Omron Sysmac Studio project ProjFinal (Sysmac Studio 1.56.0.64011, StandardProject)
(* A implementar Expedição *)

# Controller new_Controller_0: NX1P2-1040DT1 version 1.60
Units and slaves: Unit 1 : NX-ID5442 (N1); Unit 2 : NX-OD5256 (N2)
Task PrimaryTask (priority 4, period or condition 2000): Program0
Library OEN_Communication_V1_0_22 1.0.22 (contents left out)

VAR_GLOBAL
    Garra_LIDAzul_Apertar : BOOL;  (* Outputs *)
    out_dig : ARRAY[0..99] OF BOOL;
    in_dig : ARRAY[0..99] OF BOOL;
    out_analog : ARRAY[0..99] OF WORD;  (* [2] Eixo_X_Verde *)
    inp_analog : ARRAY[0..99] OF WORD;
    Requests : ARRAY[0..3] OF OEN\Modbus\sModbusReq := [(Enable := True, NodeAdr := 1, FunctionCode := Fn02_ReadDiscreteInputs, Read := (StartAddressRemote := 0, StartAddressLocal := 0, Count := 90), Write := (StartAddressRemote := 0, StartAddressLocal := 0, Count := 100)), (Enable := True, NodeAdr := 1, FunctionCode := Fn15_WriteMultipleCoils, Read := (StartAddressRemote := 0, StartAddressLocal := 0, Count := 100), Write := (StartAddressRemote := 0, StartAddressLocal := 0, Count := 95)), (Enable := True, NodeAdr := 1, FunctionCode := Fn04_ReadInputRegisters, Read := (StartAddressRemote := 0, StartAddressLocal := 0, Count := 50), Write := (StartAddressRemote := 0, StartAddressLocal := 0, Count := 100)), (Enable := True, NodeAdr := 1, FunctionCode := Fn16_WriteMultipleRegisters, Read := (StartAddressRemote := 0, StartAddressLocal := 0, Count := 0), Write := (StartAddressRemote := 0, StartAddressLocal := 0, Count := 50))];
END_VAR
VAR_GLOBAL RETAIN
    Sensor_X_Inicial AT %D33.05 : BOOL;  (* Inputs *)
    Passadeira_2_BaseVerde AT %D18.03 : BOOL;  (* Outputs *)
    Eixo_X_LIDVerde AT %D17.07 : BOOL;  (* Outputs *)
    Sensor_Z_LID_Verde AT %D9.00 : BOOL;  (* Inputs *)
    Botao_START AT %D7.00 : BOOL;  (* Inputs *)
    Botao_RESET AT %D7.02 : BOOL;  (* Inputs *)
END_VAR
VAR_GLOBAL
    Botao_Emergencia : BOOL;  (* Inputs *)
END_VAR
VAR_GLOBAL RETAIN
    Botao_STOP AT %D7.01 : BOOL;  (* Inputs *)
    Sensor_Presença_Inicial AT %D33.00 : BOOL;  (* Inputs *)
    Sensor_Garra_Apertar_Inicial AT %D33.07 : BOOL;  (* Inputs *)
    Sensor_Garra_Levantar_Inicial AT %D33.08 : BOOL;  (* Inputs *)
    Sensor_Succao_Inicial AT %D33.03 : BOOL;  (* Inputs *)
    Sensor_Rodar_Inicial AT %D33.04 : BOOL;  (* Inputs *)
END_VAR
VAR_GLOBAL
    Sensor_LIDS_Inicial : BOOL;  (* Inputs *)
END_VAR
VAR_GLOBAL RETAIN
    Sensor_CNC AT %D33.02 : BOOL;  (* Inputs *)
    Sensor_Presenca_LIDS_Geral AT %D33.01 : BOOL;  (* Inputs *)
END_VAR
VAR_GLOBAL
    Sensor_Presenca_LIDS_Verde : BOOL;  (* Inputs *)
    Sensor_Presenca_LIDS_Azul : BOOL;  (* Inputs *)
END_VAR
VAR_GLOBAL RETAIN
    Sensor_Garra_Apertar_LID_Azul AT %D8.01 : BOOL;  (* Inputs *)
    Sensor_Garra_Apertar_LID_Verde AT %D8.00 : BOOL;  (* Inputs *)
    Fim_Curso_Garra_LID_Verde AT %D8.02 : BOOL;  (* Inputs *)
    Fim_Curso_Garra_LID_Azul AT %D8.03 : BOOL;  (* Inputs *)
    Sensor_Z_LID_Azul AT %D9.01 : BOOL;  (* Inputs *)
    Sensor_X_LID_Verde AT %D9.02 : BOOL;  (* Inputs *)
    Sensor_X_LID_Azul AT %D9.03 : BOOL;  (* Inputs *)
    Sensor_Succao_LID_Verde AT %D9.04 : BOOL;  (* Inputs *)
    Sensor_Succao_LID_Azul AT %D9.05 : BOOL;  (* Inputs *)
    Sensor_Rodar_Gripper_LID_Verde AT %D9.06 : BOOL;  (* Inputs *)
    Sensor_Rodar_Gripper_LID_Azul AT %D9.07 : BOOL;  (* Inputs *)
    Sensor_Rodar_LID_Verde AT %D9.08 : BOOL;  (* Inputs *)
    Sensor_Rodar_LID_Azul AT %D9.09 : BOOL;  (* Inputs *)
END_VAR
VAR_GLOBAL
    Sensor_Presenca_Integracao_LIDVerde : BOOL;  (* Inputs *)
    Sensor_Presenca_Integracao_LIDAzul : BOOL;  (* Inputs *)
    Sensor_Presenca_Bases : BOOL;  (* Inputs *)
    Sensor_Presenca_BaseVerde : BOOL;  (* Inputs *)
    Sensor_Presenca_BaseAzul : BOOL;  (* Inputs *)
END_VAR
VAR_GLOBAL RETAIN
    Sensor_Garra_Apertar_BaseVerde AT %D14.00 : BOOL;  (* Inputs *)
    Sensor_Garra_Apertar_BaseAzul AT %D14.01 : BOOL;  (* Inputs *)
    Emitter_Inicial AT %D16.00 : BOOL;  (* Outputs *)
    Passadeira_Inicial AT %D16.01 : BOOL;  (* Outputs *)
END_VAR
VAR_GLOBAL
    Luz_Emergencia : BOOL;  (* Outputs *)
END_VAR
VAR_GLOBAL RETAIN
    Garra_Inicial_Apertar AT %D16.02 : BOOL;  (* Outputs *)
    Garra_Inicial_Levantar AT %D16.03 : BOOL;  (* Outputs *)
    Succao_Inicial AT %D16.04 : BOOL;  (* Outputs *)
    Rotacao_Inicial_CW AT %D16.05 : BOOL;  (* Outputs *)
    Rotacao_Inicial_CCW AT %D16.06 : BOOL;  (* Outputs *)
    Botao_CNC AT %D16.11 : BOOL;  (* Outputs *)
END_VAR
VAR_GLOBAL
    Garra_LIDVerde_Apertar : BOOL;  (* Outputs *)
    Garra_LIDVerde_Levantar : BOOL;  (* Outputs *)
    Garra_LIDAzul_Levantar : BOOL;  (* Outputs *)
END_VAR
VAR_GLOBAL RETAIN
    Eixo_X_LIDAzul AT %D17.08 : BOOL;  (* Outputs *)
    Eixo_Z_LIDVerde AT %D17.09 : BOOL;  (* Outputs *)
    Eixo_Z_LIDAzul AT %D17.10 : BOOL;  (* Outputs *)
    Succao_LIDVerde AT %D17.11 : BOOL;  (* Outputs *)
    Succao_LIDAzul AT %D17.12 : BOOL;  (* Outputs *)
    Rodar_Gripper_LIDVerde AT %D17.13 : BOOL;  (* Outputs *)
    Rodar_Gripper_LIDAzul AT %D17.14 : BOOL;  (* Outputs *)
    Rodar_CCW_LIDVerde AT %D17.15 : BOOL;  (* Outputs *)
    Rodar_CCW_LIDAzul AT %D18.00 : BOOL;  (* Outputs *)
    Rodar_CW_LIDVerde AT %D18.01 : BOOL;  (* Outputs *)
    Rodar_CW_LIDAzul AT %D18.02 : BOOL;  (* Outputs *)
    Passadeira_2_BaseAzul AT %D18.04 : BOOL;  (* Outputs *)
    Braço_Verde AT %D19.02 : BOOL;  (* Outputs *)
    Braço_Azul AT %D19.04 : BOOL;  (* Outputs *)
    Passadeira_1_BaseVerde AT %D19.06 : BOOL;  (* Outputs *)
    Passadeira_1_BaseAzul AT %D19.07 : BOOL;  (* Outputs *)
    Garra_BaseVerde_Apertar AT %D28.00 : BOOL;  (* Outputs *)
    Garra_BaseAzul_Apertar AT %D28.01 : BOOL;  (* Outputs *)
END_VAR
VAR_GLOBAL
    Luz_LIDVerde : BOOL;  (* Outputs *)
    Luz_LIDAzul : BOOL;  (* Outputs *)
    Luz_BaseVerde : BOOL;  (* Outputs *)
    Luz_BaseAzul : BOOL;  (* Outputs *)
END_VAR
VAR_GLOBAL RETAIN
    Sensor_Z_Inicial AT %D33.06 : BOOL;  (* Inputs *)
    Eixo_X_Inicial AT %D16.07 : BOOL;  (* Outputs *)
    Eixo_Z_Inicial AT %D16.08 : BOOL;  (* Outputs *)
    Visão_Inicial AT %D10 : INT;
    Visão_LIDS AT %D11 : INT;
    Visão_Bases AT %D12 : INT;
    Passadeira_1_LIDS AT %D17.00 : BOOL;
    Passadeira_2_LIDS AT %D17.01 : BOOL;
    Passadeira_3_LIDS AT %D17.02 : BOOL;
    Passadeira_1_Geral AT %D19.00 : BOOL;
    Passadeira_2_Geral AT %D19.01 : BOOL;
    Passadeira_Braço_Verde AT %D19.03 : BOOL;
    Passadeira_Braço_Azul AT %D19.05 : BOOL;
END_VAR
VAR_GLOBAL
    Eixo_X_Verde : REAL;
    Eixo_Z_Verde : REAL;
END_VAR
VAR_GLOBAL RETAIN
    Succao_Verde AT %D28.04 : BOOL;
    Rotacao_CCW_Verde AT %D28.06 : BOOL;
    Rotacao_CW_Verde AT %D28.08 : BOOL;
END_VAR
VAR_GLOBAL
    Eixo_X_Azul : REAL;
    Eixo_Z_Azul : REAL;
END_VAR
VAR_GLOBAL RETAIN
    Succao_Azul AT %D28.05 : BOOL;
    Rotacao_CCW_Azul AT %D28.07 : BOOL;
    Rotacao_CW_Azul AT %D28.09 : BOOL;
    Sensor_Succao_Verde AT %D14.02 : BOOL;
    Sensor_Succao_Azul AT %D14.03 : BOOL;
END_VAR
VAR_GLOBAL
    Sensor_X_Verde : REAL;
    Sensor_Z_Verde : REAL;
    Sensor_X_Azul : REAL;
    Sensor_Z_Azul : REAL;
END_VAR
VAR_GLOBAL RETAIN
    Sensor_Rodar_Verde AT %D14.06 : BOOL;
    Sensor_Rodar_Azul AT %D14.07 : BOOL;
END_VAR
VAR_GLOBAL
    etapas_integração : INT;
    etapas_lids : INT;
    etapas_bases : INT;
    etapas_separaçãoinicial : INT;
    etapas_organização : INT;
    etapas_main : INT;
END_VAR
VAR_GLOBAL RETAIN
    Curva_Rolos_Verde AT %D29.04 : BOOL;
    Rolos_Verde_1 AT %D29.01 : BOOL;
    Rolos_Verde_2 AT %D29.02 : BOOL;
    Rolos_Verde_3 AT %D29.03 : BOOL;
    Garra_Direita_Verde AT %D29.07 : BOOL;
    Garra_Esquerda_Verde AT %D29.05 : BOOL;
    Levantar_Empilhador_Verde AT %D29.06 : BOOL;
    Sensor_Presença_PeçasVerdes AT %D15.00 : BOOL;
    FC_Meio_Verde AT %D15.01 : BOOL;
    FC_Esquerdo_Verde AT %D15.02 : BOOL;
    FC_Direito_Verde AT %D15.03 : BOOL;
    Sensor_Levantar_Empilhador_Verde AT %D15.04 : BOOL;
    Conta_Empi_Verde AT %D25 : INT;
    Sensor_Posição_Empi_Verde AT %D15.05 : BOOL;
END_VAR
VAR_GLOBAL
    Contador_Lid_Verde : INT;
    Contador_Base_Azul : INT;
    Contador_Base_Verde : INT;
END_VAR
VAR_GLOBAL RETAIN
    Removedor_Bases AT %D19.08 : BOOL;
END_VAR
VAR_GLOBAL
    Contador_LID_Azul : INT;
END_VAR
VAR_GLOBAL RETAIN
    Removedor_LIDS AT %D18.05 : BOOL;
END_VAR
VAR_GLOBAL
    Contador_Integradas_Verde : INT;
    Contador_Integradas_Azul : INT;
END_VAR
VAR_GLOBAL RETAIN
    Flag_LIDS_Azul : BOOL;
    Sensor_Base_Azul AT %D13.02 : BOOL;
    Sensor_Base_Verde AT %D13.01 : BOOL;
    Flag_Integração_Azul : BOOL;
    Rolos_Azul_1 AT %D29.09 : BOOL;
    Curva_Rolos_Azul AT %D29.10 : BOOL;
    Rolos_Azul_2 AT %D29.11 : BOOL;
    Rolos_Azul_3 AT %D29.12 : BOOL;
    Garra_Esquerda_Azul AT %D29.13 : BOOL;
    Garra_Direita_Azul AT %D29.14 : BOOL;
    Levantar_Empilhador_Azul AT %D29.15 : BOOL;
    Emitter_CPVerde AT %D29.00 : BOOL;
    Emitter_CPAzul AT %D29.08 : BOOL;
    Sensor_Presença_PeçasAzuis AT %D15.06 : BOOL;
    FC_Meio_Azul AT %D15.07 : BOOL;
    FC_Esquerdo_Azul AT %D15.08 : BOOL;
    FC_Direito_Azul AT %D15.09 : BOOL;
    Sensor_Levantar_Empilhador_Azul AT %D15.10 : BOOL;
    Sensor_Posicao_Empi_Azul AT %D15.11 : BOOL;
    Conta_Empi_Azul AT %D24 : INT;
    Flag_Integração_Verde : BOOL;
    Flag_LIDS_Verde : BOOL;
    Sensor_Bases AT %D13.00 : BOOL;
END_VAR
VAR_GLOBAL
    LED_Verde : BOOL;
    LED_Vermelho : BOOL;
    Flag_Botão_STOP_SI : BOOL;
    Flag_Botao_STOP_B : BOOL;
    Flag_Botao_STOP_L : BOOL;
    Flag_Botao_STOP_I : BOOL;
    Flag_Botao_Stop_O : BOOL;
    Flag_Emergência : BOOL;
    Reset_Factory : BOOL;
    IN_BIT_01 : BOOL;  (* BOTAO START; at BuiltInIO://cpu/#0/Input_Bit_01 *)
    IN_BIT_02 : BOOL;  (* BOTAO STOP; at BuiltInIO://cpu/#0/Input_Bit_02 *)
    OUT_BIT_01 : BOOL;  (* LED VERMELHO; at BuiltInIO://cpu/#0/Output_Bit_01 *)
    OUT_BIT_02 : BOOL;  (* LED VERDE; at BuiltInIO://cpu/#0/Output_Bit_02 *)
    IN_BIT_03 : BOOL;  (* BOTAO EMERGENCIA; at BuiltInIO://cpu/#0/Input_Bit_03 *)
END_VAR
VAR_GLOBAL RETAIN
    Sensor_LID_Verde AT %D8.04 : BOOL;
    Sensor_LID_Azul AT %D8.05 : BOOL;
END_VAR
VAR_GLOBAL
    Flag_Integração_LIDVerde : BOOL;
    Flag_Integração_LIDAzul : BOOL;
END_VAR
VAR_GLOBAL RETAIN
    Sensor_Garra_Apertar_IntLIDVerde AT %D14.04 : BOOL;
    Sensor_Garra_Apertar_IntLIDAzul AT %D14.05 : BOOL;
    Garra_LIDVerdeInt_apertar AT %D28.02 : BOOL;
    Garra_LIDAzulInt_apertar AT %D28.03 : BOOL;
    Garra_LIDAzul_Levant AT %D17.06 : BOOL;
    Garra_LIDVerde_Levant AT %D17.05 : BOOL;
    Garra_LIDAzul_Apert AT %D17.04 : BOOL;
    Garra_LIDVerde_Apert AT %D17.03 : BOOL;
    Expedição_Caixas_Verdes AT %D26 : INT;
    Expedição_Caixas_Azuis AT %D27 : INT;
END_VAR
VAR_GLOBAL
    etapas_expediçãoazul : INT;
    Rolos_Exp_Azul_1 : BOOL;
    Rolos_Exp_Azul_2 : BOOL;
    Remover_Exp_Azul : BOOL;
    Emitter_Exp_Azul : BOOL;
    Rolos_Exp_Azul_3 : BOOL;
    Remover_Caixa_Azul : BOOL;
    etapas_expediçãoverde : INT;
    Rolos_Exp_Verde_1 : BOOL;
    Remover_Exp_Verde : BOOL;
    Emitter_Exp_Verde : BOOL;
    Remover_Caixa_Verde : BOOL;
    Rolos_Exp_Verde_2 : BOOL;
    Levantar_Empilhador_Azul_Expedição : BOOL;
    Garra_Direita_Azul_Expedição : BOOL;
    Levantar_Empilhador_Verde_Expedição : BOOL;
    Garra_Direita_Verde_Expedição : BOOL;
END_VAR
VAR_GLOBAL RETAIN
    Stock_Azul : INT;
    Stock_Verde : INT;
    Nº_Caixas_Expedidas_Azuis AT %D22 : INT;
    Nº_Caixas_Expedidas_Verdes AT %D23 : INT;
END_VAR
VAR_GLOBAL
    Flag_Botao_Stop_EA : BOOL;
    Flag_Botao_Stop_EV : BOOL;
END_VAR
VAR_GLOBAL RETAIN
    SI_LED AT %D7.02 : BOOL;
    L_LED AT %D7.03 : BOOL;
    B_LED AT %D7.04 : BOOL;
    I_LED AT %D7.05 : BOOL;
    A_LED AT %D7.06 : BOOL;
    E_LED AT %D7.07 : BOOL;
    Peças_Integradas_Verdes_HMI AT %D20 : INT;
    Peças_Integradas_Azuis_HMI AT %D21 : INT;
    Pusher AT %D16.09 : BOOL;
    Remove_Peças_Más AT %D16.10 : BOOL;
END_VAR
VAR_GLOBAL
    FC_Traseiro_Pusher : BOOL;
END_VAR
VAR_GLOBAL RETAIN
    Eixo_X_Verde_HMI AT %D40 : INT;
    Eixo_X_Azul_HMI AT %D41 : INT;
    Eixo_Z_Verde_HMI AT %D42 : INT;
    Eixo_Z_Azul_HMI AT %D43 : INT;
END_VAR

PROGRAM Program0
VAR
    TCP_CLIENT : OEN\Modbus\ModbusTCP_Client;
    TimerIntegraçãoAzul : TON;
    TimerIntegraçãoAzul2 : TON;
    TimerIntegraçãoAzul3 : TON;
    TimerIntegraçãoAzul4 : TON;
    TimerIntegraçãoVerde : TON;
    TimerIntegraçãoVerde2 : TON;
    TimerIntegraçãoVerde3 : TON;
    TimerIntegraçãoVerde4 : TON;
    TimerSensorEmpiVerde : TON;
    TON_EMPVERDE1 : TON;
    TON_EMPVERDE2 : TON;
    TON_EMPVERDE3 : TON;
    TON_EMPVERDE4 : TON;
    TimerSensorEmpiAzul : TON;
    TON_EMPAZUL1 : TON;
    TON_EMPAZUL2 : TON;
    TON_EMPAZUL3 : TON;
    TON_EMPAZUL4 : TON;
    Timer_Gripper_Verde : TON;
    LIDVerde1 : TON;
    LIDVerde2 : TON;
    Timer_Gripper_Azul : TON;
    LIDAzul1 : TON;
    LIDAzul2 : TON;
    TimerRemovedorBases : TON;
    Timer_Base_Verde : TON;
    Timer_Base_Azul : TON;
    TimerPickNPlace : TON;
    Timer_LidVerde_Garra : TON;
    Timer_LidAzul_Garra : TON;
    TimerRemovedorLIDS : TON;
    CTUEmpiVerde : CTU;
    CTUEmpiAzul : CTU;
    CTUIntegradasVerde : CTU;
    CTUIntegradasAzul : CTU;
    CTULidVerde : CTU;
    CTULidAzul : CTU;
    CTUBaseVerde : CTU;
    CTUBaseAzul : CTU;
    Teste : TON;
    Timer_LID_Verde : TON;
    Timer_LID_Azul : TON;
    Timer_Expedição_Azul : TON;
    TON_EMPAZUL5 : TON;
    TON_EMPAZUL6 : TON;
    TON_EMPAZUL7 : TON;
    TON_EMPAZUL8 : TON;
    TON_EMPAZUL9 : TON;
    TON_EMPAZUL10 : TON;
    TON_EMPAZUL11 : TON;
    CTD_Empi_Azul : CTD;
    CTD_Restante_Exp_Azul : CTD;
    TON_EMPVERDE5 : TON;
    TON_EMPVERDE6 : TON;
    TON_EMPVERDE7 : TON;
    TON_EMPVERDE8 : TON;
    TON_EMPVERDE9 : TON;
    TON_EMPVERDE10 : TON;
    TON_EMPVERDE11 : TON;
    TON_EMPAZUL12 : TON;
    TON_EMPVERDE12 : TON;
    CTD_Stock_Azul : CTD;
    TON_COUNTERSAZUL : TON;
    TIMERFLAGS : TON;
    TRIGSUBS : R_TRIG;
    TRIGSUBS1 : R_TRIG;
    TRIGSUB2 : R_TRIG;
    TRIGLIDA1 : R_TRIG;
    TRIGLIDV1 : R_TRIG;
    TRIGBASEA1 : R_TRIG;
    TRIGBASEV1 : R_TRIG;
    TRIGINTEGRADAV1 : R_TRIG;
    TRIGINTEGRADAA1 : R_TRIG;
    TRIGEMPV1 : R_TRIG;
    TRIGEMPA1 : R_TRIG;
    TRIGSUBS2 : R_TRIG;
    TRIGEXPVERDE1 : R_TRIG;
    TRIGEXPVERDE2 : R_TRIG;
    TRIGEXPVERDE3 : R_TRIG;
END_VAR
VAR RETAIN
    Emitter_Inicial_HMI AT %D0.00 : BOOL;
    Passadeira_Inicial_HMI AT %D0.01 : BOOL;
    Garra_Inicial_Apertar_HMI AT %D0.02 : BOOL;
    Garra_Inicial_Levantar_HMI AT %D0.03 : BOOL;
    Succao_Inicial_HMI AT %D0.04 : BOOL;
    Rotação_Inicial_CW_HMI AT %D0.05 : BOOL;
    Rotacao_Inicial_CCW_HMI AT %D0.06 : BOOL;
    Eixo_X_Inicial_HMI AT %D0.07 : BOOL;
    Eixo_Z_Inicial_HMI AT %D0.08 : BOOL;
    Botao_CNC_HMI AT %D0.09 : BOOL;
    Passadeira_1_LIDS_HMI AT %D1.00 : BOOL;
    Passadeira_2_LIDS_HMI AT %D1.01 : BOOL;
    Passadeira_3_LIDS_HMI AT %D1.02 : BOOL;
    Passadeira_2_BaseVerde_HMI AT %D1.03 : BOOL;
    Passadeira_2_BaseAzul_HMI AT %D1.04 : BOOL;
    Garra_LIDVerde_Apert_HMI AT %D1.05 : BOOL;
    Garra_LIDAzul_Apert_HMI AT %D1.06 : BOOL;
    Garra_LIDVerde_Levant_HMI AT %D1.07 : BOOL;
    Garra_LIDAzul_Levant_HMI AT %D1.08 : BOOL;
    Removedor_LIDS_HMI AT %D1.09 : BOOL;
    Eixo_X_LIDVerde_HMI AT %D2.00 : BOOL;
    Eixo_X_LIDAzul_HMI AT %D2.01 : BOOL;
    Eixo_Z_LID_Verde_HMI AT %D2.02 : BOOL;
    Eixo_Z_LIDAzul_HMI AT %D2.03 : BOOL;
    Succao_LIDVerde_HMI AT %D2.04 : BOOL;
    Succao_LIDAzul_HMI AT %D2.05 : BOOL;
    Rodar_Gripper_LIDVerde_HMI AT %D2.06 : BOOL;
    Rodar_Gripper_LIDAzul_HMI AT %D2.07 : BOOL;
    Rodar_CCW_LIDVerde_HMI AT %D2.08 : BOOL;
    Rodar_CCW_LIDAzul_HMI AT %D2.09 : BOOL;
    Rodar_CW_LIDVerde_HMI AT %D2.10 : BOOL;
    Rodar_CW_LIDAzul_HMI AT %D2.11 : BOOL;
    Passadeira_1_Geral_HMI AT %D3.00 : BOOL;
    Passadeira_2_Geral_HMI AT %D3.01 : BOOL;
    Braço_Verde_HMI AT %D3.02 : BOOL;
    Passadeira_Braço_Verde_HMI AT %D3.03 : BOOL;
    Braço_Azul_HMI AT %D3.04 : BOOL;
    Passadeira_Braço_Azul_HMI AT %D3.05 : BOOL;
    Passadeira_1_BaseVerde_HMI AT %D3.06 : BOOL;
    Passadeira_1_BaseAzul_HMI AT %D3.07 : BOOL;
    Removedor_Bases_HMI AT %D3.08 : BOOL;
    Garra_BaseAzul_Apertar_HMI AT %D4.00 : BOOL;
    Garra_BaseVerde_Apertar_HMI AT %D4.01 : BOOL;
    Garra_LIDVerdeInt_apertar_HMI AT %D4.02 : BOOL;
    Garra_LIDAzulInt_apertar_HMI AT %D4.03 : BOOL;
    Succao_Verde_HMI AT %D4.04 : BOOL;
    Succao_Azul_HMI AT %D4.05 : BOOL;
    Rotacao_CCW_Verde_HMI AT %D4.06 : BOOL;
    Rotacao_CCW_Azul_HMI AT %D4.07 : BOOL;
    Rotacao_CW_Verde_HMI AT %D4.08 : BOOL;
    Rotacao_CW_Azul_HMI AT %D4.09 : BOOL;
    Emitter_CPVerde_HMI AT %D5.00 : BOOL;
    Rolos_Verde_1_HMI AT %D5.01 : BOOL;
    Rolos_Verde_2_HMI AT %D5.02 : BOOL;
    Rolos_Verde_3_HMI AT %D5.03 : BOOL;
    Curva_Rolos_Verde_HMI AT %D5.04 : BOOL;
    Emitter_CPAzul_HMI AT %D5.05 : BOOL;
    Rolos_Azul_1_HMI AT %D5.06 : BOOL;
    Curva_Rolos_Azul_HMI AT %D5.07 : BOOL;
    Rolos_Azul_2_HMI AT %D5.08 : BOOL;
    Rolos_Azul_3_HMI AT %D5.09 : BOOL;
    Garra_Esquerda_Azul_HMI AT %D6.00 : BOOL;
    Garra_Direita_Azul_HMI AT %D6.01 : BOOL;
    Levantar_Empilhador_Azul_HMI AT %D6.02 : BOOL;
    Garra_Esquerda_Verde_HMI AT %D6.03 : BOOL;
    Levantar_Empilhador_Verde_HMI AT %D6.04 : BOOL;
    Garra_Direita_Verde_HMI AT %D6.05 : BOOL;
END_VAR
VAR
    TRIGINTEGRADAA2 : R_TRIG;
    TRIGINTEGRADAV2 : R_TRIG;
    TON_Peça_Máe : TON;
    TON_Peça_Má : TON;
END_VAR
VAR RETAIN
    Pusher_HMI AT %D0.10 : BOOL;
    Remove_Peças_Más_HMI AT %D0.11 : BOOL;
END_VAR
VAR
    RESETTON : TON;
END_VAR
VAR_EXTERNAL
    Emitter_Inicial : BOOL;
    Garra_Inicial_Apertar : BOOL;
    Garra_Inicial_Levantar : BOOL;
    Braço_Azul : BOOL;
    Braço_Verde : BOOL;
    in_dig : ARRAY[0..99] OF BOOL;
    out_dig : ARRAY[0..99] OF BOOL;
    out_analog : ARRAY[0..99] OF WORD;
    Requests : ARRAY[0..3] OF OEN\Modbus\sModbusReq;
    Botao_RESET : BOOL;
    Botao_Emergencia : BOOL;
    Botao_START : BOOL;
    Botao_STOP : BOOL;
    Luz_Emergencia : BOOL;
    Passadeira_Inicial : BOOL;
    Sensor_Presença_Inicial : BOOL;
    Sensor_Garra_Apertar_Inicial : BOOL;
    Sensor_Garra_Levantar_Inicial : BOOL;
    Sensor_CNC : BOOL;
    Sensor_Succao_Inicial : BOOL;
    Sensor_Z_Inicial : BOOL;
    Sensor_X_Inicial : BOOL;
    Sensor_Rodar_Inicial : BOOL;
    Sensor_LIDS_Inicial : BOOL;
    Sensor_Presenca_LIDS_Geral : BOOL;
    Sensor_Presenca_LIDS_Verde : BOOL;
    Sensor_Presenca_LIDS_Azul : BOOL;
    Botao_CNC : BOOL;
    Sensor_Garra_Apertar_LID_Azul : BOOL;
    Sensor_Garra_Apertar_LID_Verde : BOOL;
    Fim_Curso_Garra_LID_Verde : BOOL;
    Fim_Curso_Garra_LID_Azul : BOOL;
    Sensor_Z_LID_Verde : BOOL;
    Sensor_Z_LID_Azul : BOOL;
    Sensor_X_LID_Verde : BOOL;
    Sensor_X_LID_Azul : BOOL;
    Sensor_Succao_LID_Verde : BOOL;
    Sensor_Succao_LID_Azul : BOOL;
    Sensor_Rodar_Gripper_LID_Verde : BOOL;
    Sensor_Rodar_Gripper_LID_Azul : BOOL;
    Sensor_Rodar_LID_Verde : BOOL;
    Sensor_Rodar_LID_Azul : BOOL;
    Sensor_Presenca_Integracao_LIDVerde : BOOL;
    Sensor_Presenca_Integracao_LIDAzul : BOOL;
    Sensor_Presenca_Bases : BOOL;
    Sensor_Presenca_BaseVerde : BOOL;
    Sensor_Presenca_BaseAzul : BOOL;
    Sensor_Garra_Apertar_BaseVerde : BOOL;
    Sensor_Garra_Apertar_BaseAzul : BOOL;
    Succao_Inicial : BOOL;
    Rotacao_Inicial_CW : BOOL;
    Rotacao_Inicial_CCW : BOOL;
    Eixo_Z_Inicial : BOOL;
    Eixo_X_Inicial : BOOL;
    Garra_LIDVerde_Apertar : BOOL;
    Garra_LIDAzul_Apertar : BOOL;
    Garra_LIDVerde_Levantar : BOOL;
    Garra_LIDAzul_Levantar : BOOL;
    Eixo_X_LIDVerde : BOOL;
    Eixo_X_LIDAzul : BOOL;
    Eixo_Z_LIDVerde : BOOL;
    Eixo_Z_LIDAzul : BOOL;
    Succao_LIDVerde : BOOL;
    Succao_LIDAzul : BOOL;
    Rodar_Gripper_LIDVerde : BOOL;
    Rodar_Gripper_LIDAzul : BOOL;
    Rodar_CCW_LIDVerde : BOOL;
    Rodar_CCW_LIDAzul : BOOL;
    Rodar_CW_LIDVerde : BOOL;
    Rodar_CW_LIDAzul : BOOL;
    Passadeira_2_BaseVerde : BOOL;
    Passadeira_2_BaseAzul : BOOL;
    Passadeira_1_BaseVerde : BOOL;
    Passadeira_1_BaseAzul : BOOL;
    Garra_BaseVerde_Apertar : BOOL;
    Garra_BaseAzul_Apertar : BOOL;
    Luz_LIDVerde : BOOL;
    Luz_LIDAzul : BOOL;
    Luz_BaseVerde : BOOL;
    Luz_BaseAzul : BOOL;
    Visão_Inicial : INT;
    Visão_LIDS : INT;
    Visão_Bases : INT;
    Passadeira_1_LIDS : BOOL;
    Passadeira_2_LIDS : BOOL;
    Passadeira_3_LIDS : BOOL;
    Passadeira_1_Geral : BOOL;
    Passadeira_2_Geral : BOOL;
    Passadeira_Braço_Verde : BOOL;
    Passadeira_Braço_Azul : BOOL;
    Eixo_X_Verde : REAL;
    Eixo_Z_Verde : REAL;
    Succao_Verde : BOOL;
    Rotacao_CCW_Verde : BOOL;
    Rotacao_CW_Verde : BOOL;
    Eixo_X_Azul : REAL;
    Eixo_Z_Azul : REAL;
    Succao_Azul : BOOL;
    Rotacao_CCW_Azul : BOOL;
    Rotacao_CW_Azul : BOOL;
    Sensor_Succao_Verde : BOOL;
    Sensor_Succao_Azul : BOOL;
    Sensor_X_Verde : REAL;
    Sensor_Z_Verde : REAL;
    Sensor_X_Azul : REAL;
    Sensor_Z_Azul : REAL;
    Sensor_Rodar_Verde : BOOL;
    Sensor_Rodar_Azul : BOOL;
    inp_analog : ARRAY[0..99] OF WORD;
    etapas_integração : INT;
    etapas_lids : INT;
    etapas_bases : INT;
    etapas_separaçãoinicial : INT;
    etapas_organização : INT;
    etapas_main : INT;
    Curva_Rolos_Verde : BOOL;
    Rolos_Verde_1 : BOOL;
    Rolos_Verde_2 : BOOL;
    Rolos_Verde_3 : BOOL;
    Sensor_Presença_PeçasVerdes : BOOL;
    Garra_Esquerda_Verde : BOOL;
    FC_Meio_Verde : BOOL;
    FC_Esquerdo_Verde : BOOL;
    FC_Direito_Verde : BOOL;
    Levantar_Empilhador_Verde : BOOL;
    Sensor_Levantar_Empilhador_Verde : BOOL;
    Conta_Empi_Verde : INT;
    Sensor_Posição_Empi_Verde : BOOL;
    Garra_Direita_Verde : BOOL;
    Contador_Lid_Verde : INT;
    Contador_Base_Azul : INT;
    Contador_Base_Verde : INT;
    Removedor_Bases : BOOL;
    Contador_LID_Azul : INT;
    Removedor_LIDS : BOOL;
    Contador_Integradas_Verde : INT;
    Contador_Integradas_Azul : INT;
    Flag_LIDS_Azul : BOOL;
    Sensor_Base_Azul : BOOL;
    Sensor_Base_Verde : BOOL;
    Flag_Integração_Azul : BOOL;
    Rolos_Azul_1 : BOOL;
    Curva_Rolos_Azul : BOOL;
    Rolos_Azul_2 : BOOL;
    Rolos_Azul_3 : BOOL;
    Garra_Esquerda_Azul : BOOL;
    Garra_Direita_Azul : BOOL;
    Levantar_Empilhador_Azul : BOOL;
    Emitter_CPVerde : BOOL;
    Emitter_CPAzul : BOOL;
    Sensor_Presença_PeçasAzuis : BOOL;
    FC_Meio_Azul : BOOL;
    FC_Esquerdo_Azul : BOOL;
    FC_Direito_Azul : BOOL;
    Sensor_Levantar_Empilhador_Azul : BOOL;
    Sensor_Posicao_Empi_Azul : BOOL;
    Conta_Empi_Azul : INT;
    Flag_Integração_Verde : BOOL;
    Flag_LIDS_Verde : BOOL;
    Sensor_Bases : BOOL;
    LED_Verde : BOOL;
    LED_Vermelho : BOOL;
    Flag_Botão_STOP_SI : BOOL;
    Flag_Botao_STOP_B : BOOL;
    Flag_Botao_STOP_L : BOOL;
    Flag_Botao_STOP_I : BOOL;
    Flag_Botao_Stop_O : BOOL;
    Flag_Emergência : BOOL;
    Reset_Factory : BOOL;
    OUT_BIT_02 : BOOL;
    OUT_BIT_01 : BOOL;
    IN_BIT_01 : BOOL;
    IN_BIT_02 : BOOL;
    IN_BIT_03 : BOOL;
    Sensor_LID_Verde : BOOL;
    Sensor_LID_Azul : BOOL;
    Flag_Integração_LIDVerde : BOOL;
    Flag_Integração_LIDAzul : BOOL;
    Sensor_Garra_Apertar_IntLIDVerde : BOOL;
    Sensor_Garra_Apertar_IntLIDAzul : BOOL;
    Garra_LIDVerdeInt_apertar : BOOL;
    Garra_LIDAzulInt_apertar : BOOL;
    Garra_LIDAzul_Levant : BOOL;
    Garra_LIDVerde_Levant : BOOL;
    Garra_LIDAzul_Apert : BOOL;
    Garra_LIDVerde_Apert : BOOL;
    Expedição_Caixas_Verdes : INT;
    Expedição_Caixas_Azuis : INT;
    etapas_expediçãoazul : INT;
    Rolos_Exp_Azul_1 : BOOL;
    Rolos_Exp_Azul_2 : BOOL;
    Remover_Exp_Azul : BOOL;
    Emitter_Exp_Azul : BOOL;
    Rolos_Exp_Azul_3 : BOOL;
    Remover_Caixa_Azul : BOOL;
    etapas_expediçãoverde : INT;
    Rolos_Exp_Verde_1 : BOOL;
    Remover_Exp_Verde : BOOL;
    Emitter_Exp_Verde : BOOL;
    Remover_Caixa_Verde : BOOL;
    Rolos_Exp_Verde_2 : BOOL;
    Levantar_Empilhador_Azul_Expedição : BOOL;
    Garra_Direita_Azul_Expedição : BOOL;
    Levantar_Empilhador_Verde_Expedição : BOOL;
    Garra_Direita_Verde_Expedição : BOOL;
    Stock_Azul : INT;
    Stock_Verde : INT;
    Nº_Caixas_Expedidas_Azuis : INT;
    Nº_Caixas_Expedidas_Verdes : INT;
    Flag_Botao_Stop_EA : BOOL;
    Flag_Botao_Stop_EV : BOOL;
    SI_LED : BOOL;
    L_LED : BOOL;
    B_LED : BOOL;
    I_LED : BOOL;
    A_LED : BOOL;
    E_LED : BOOL;
    Peças_Integradas_Verdes_HMI : INT;
    Peças_Integradas_Azuis_HMI : INT;
    Pusher : BOOL;
    Remove_Peças_Más : BOOL;
    FC_Traseiro_Pusher : BOOL;
    Eixo_X_Verde_HMI : INT;
    Eixo_X_Azul_HMI : INT;
    Eixo_Z_Verde_HMI : INT;
    Eixo_Z_Azul_HMI : INT;
END_VAR
VAR
    _p1 : BOOL;
    _p2 : BOOL;
    _p3 : BOOL;
    _p4 : BOOL;
    _p5 : BOOL;
    _p6 : BOOL;
    _p7 : BOOL;
    _p8 : BOOL;
    _p9 : BOOL;
    _p10 : BOOL;
    _p11 : BOOL;
    _p12 : BOOL;
    _p13 : BOOL;
    _p14 : BOOL;
    _p15 : BOOL;
END_VAR

(* Section ModBusComm: ladder, written here as Structured Text *)

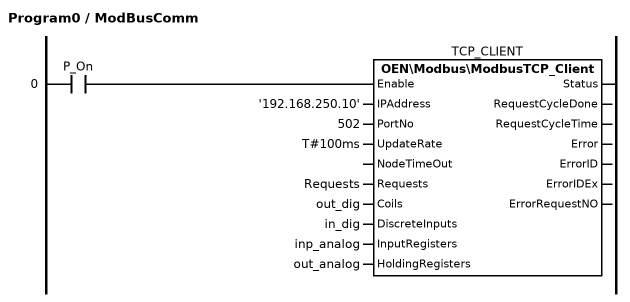
(* Rung 0 *)
TCP_CLIENT(Enable := P_On, IPAddress := '192.168.250.10', PortNo := 502, UpdateRate := T#100ms, Requests := Requests, Coils := out_dig, DiscreteInputs := in_dig, InputRegisters := inp_analog, HoldingRegisters := out_analog);

(* Section Main_Etapas: ladder, written here as Structured Text *)

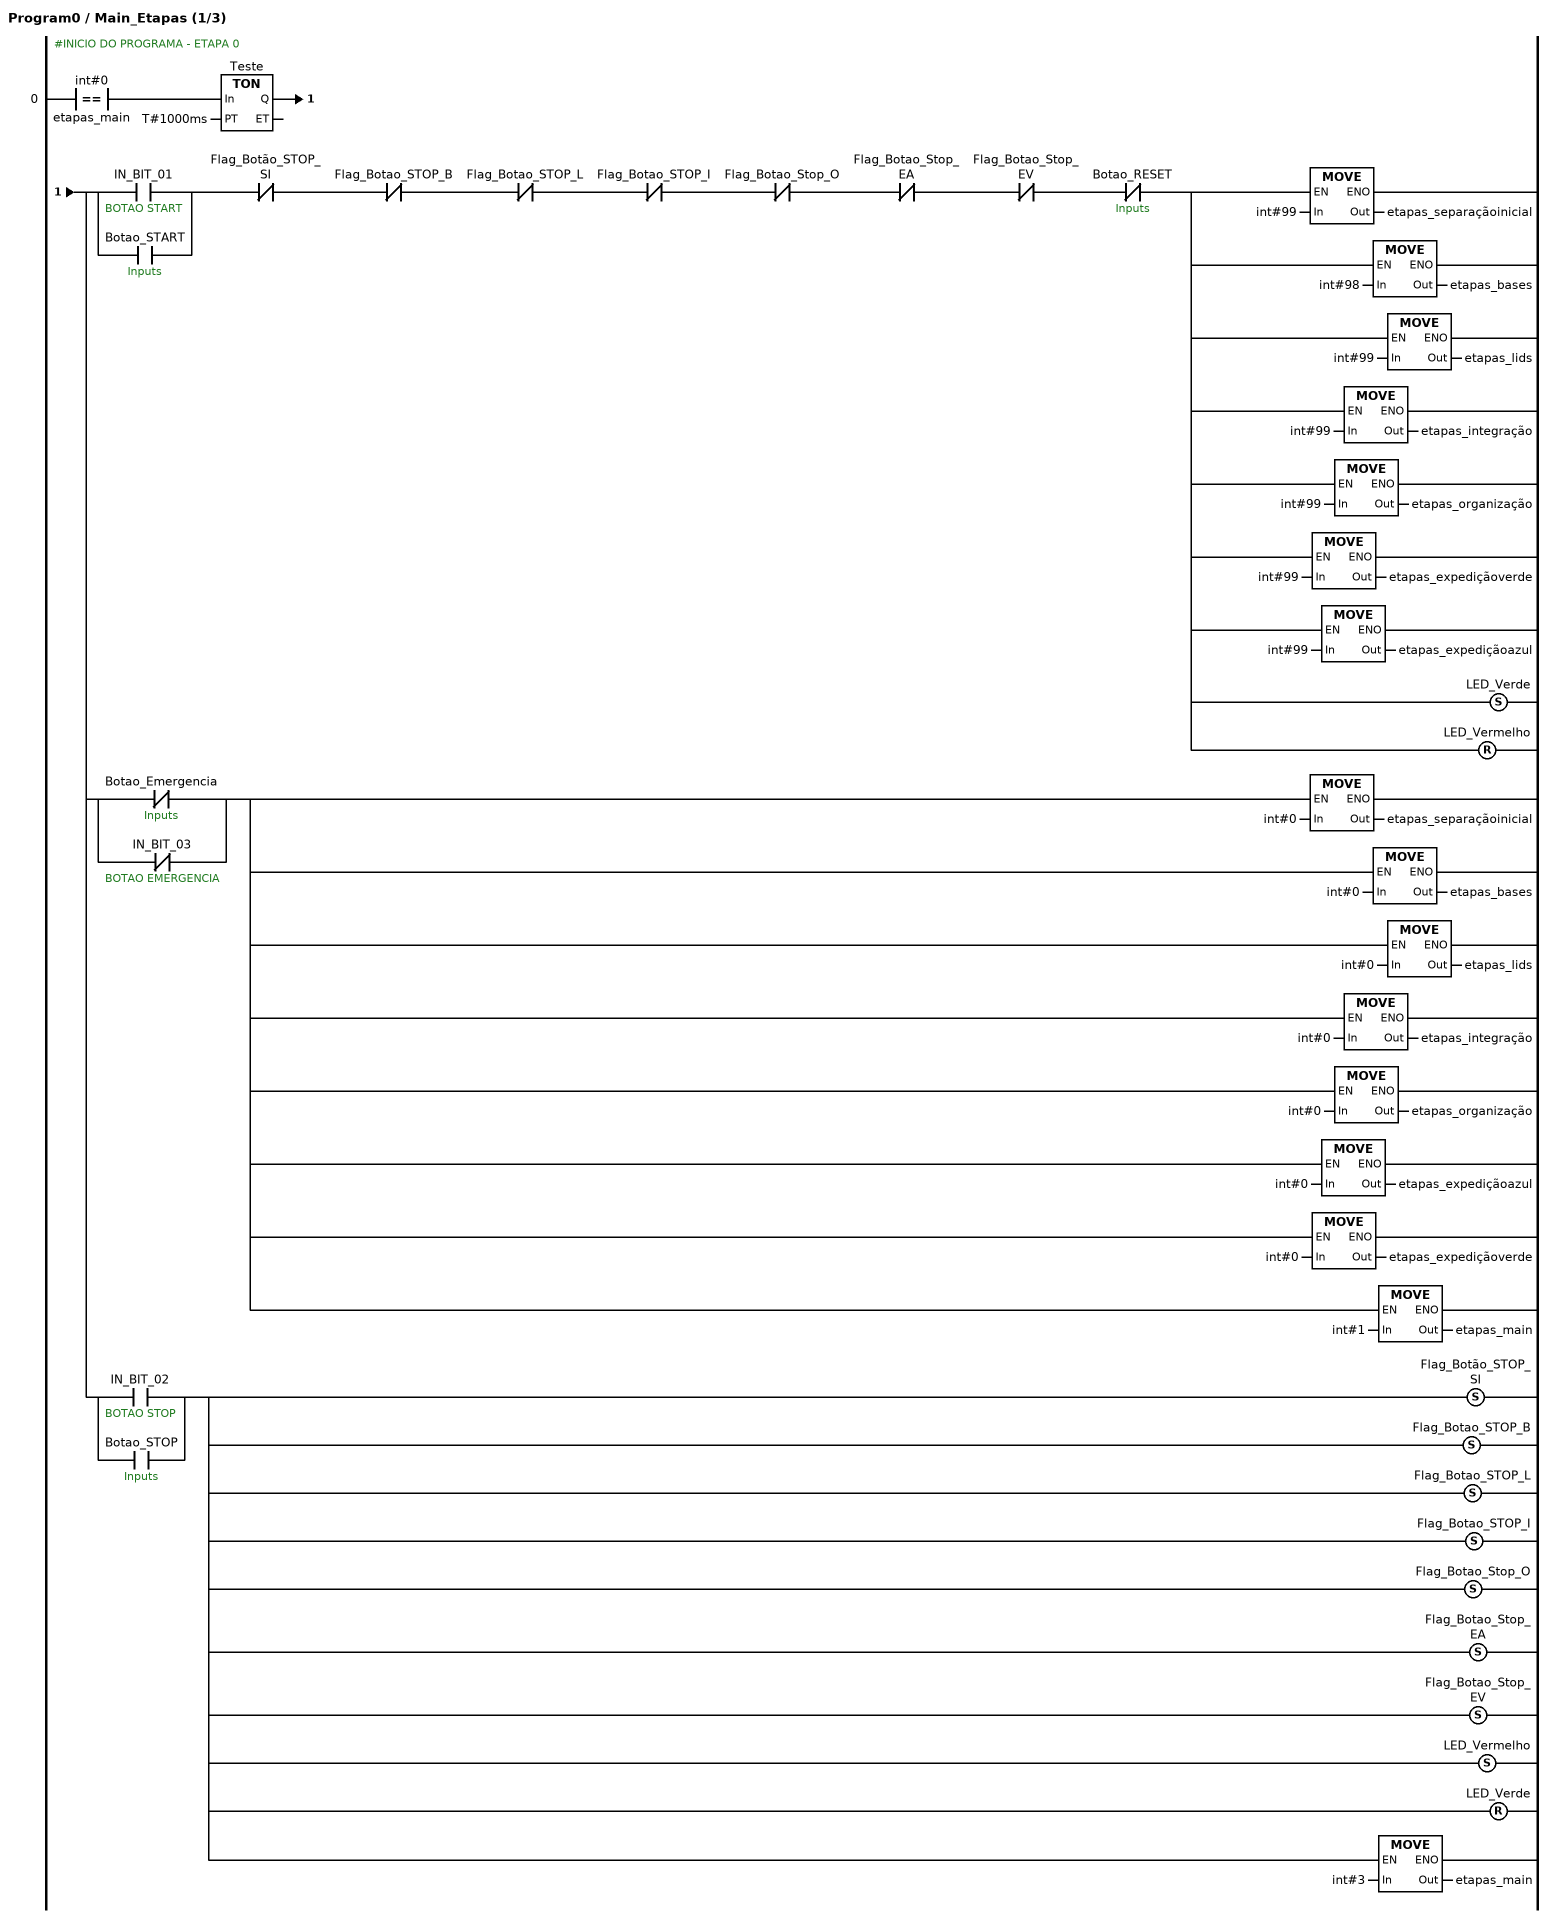
(* Rung 0: #INICIO DO PROGRAMA - ETAPA 0 *)
Teste(In := int#0 = etapas_main, PT := T#1000ms);
_p1 := Teste.Q AND (IN_BIT_01 OR Botao_START) AND NOT Flag_Botão_STOP_SI AND NOT Flag_Botao_STOP_B AND NOT Flag_Botao_STOP_L AND NOT Flag_Botao_STOP_I AND NOT Flag_Botao_Stop_O AND NOT Flag_Botao_Stop_EA AND NOT Flag_Botao_Stop_EV AND NOT Botao_RESET;
IF _p1 THEN
    etapas_separaçãoinicial := int#99;
    etapas_bases := int#98;
    etapas_lids := int#99;
    etapas_integração := int#99;
    etapas_organização := int#99;
    etapas_expediçãoverde := int#99;
    etapas_expediçãoazul := int#99;
    LED_Verde := TRUE;
    LED_Vermelho := FALSE;
END_IF;
_p2 := Teste.Q AND (NOT Botao_Emergencia OR NOT IN_BIT_03);
IF _p2 THEN
    etapas_separaçãoinicial := int#0;
    etapas_bases := int#0;
    etapas_lids := int#0;
    etapas_integração := int#0;
    etapas_organização := int#0;
    etapas_expediçãoazul := int#0;
    etapas_expediçãoverde := int#0;
    etapas_main := int#1;
END_IF;
IF Teste.Q AND (IN_BIT_02 OR Botao_STOP) THEN
    Flag_Botão_STOP_SI := TRUE;
    Flag_Botao_STOP_B := TRUE;
    Flag_Botao_STOP_L := TRUE;
    Flag_Botao_STOP_I := TRUE;
    Flag_Botao_Stop_O := TRUE;
    Flag_Botao_Stop_EA := TRUE;
    Flag_Botao_Stop_EV := TRUE;
    LED_Vermelho := TRUE;
    LED_Verde := FALSE;
    etapas_main := int#3;
END_IF;

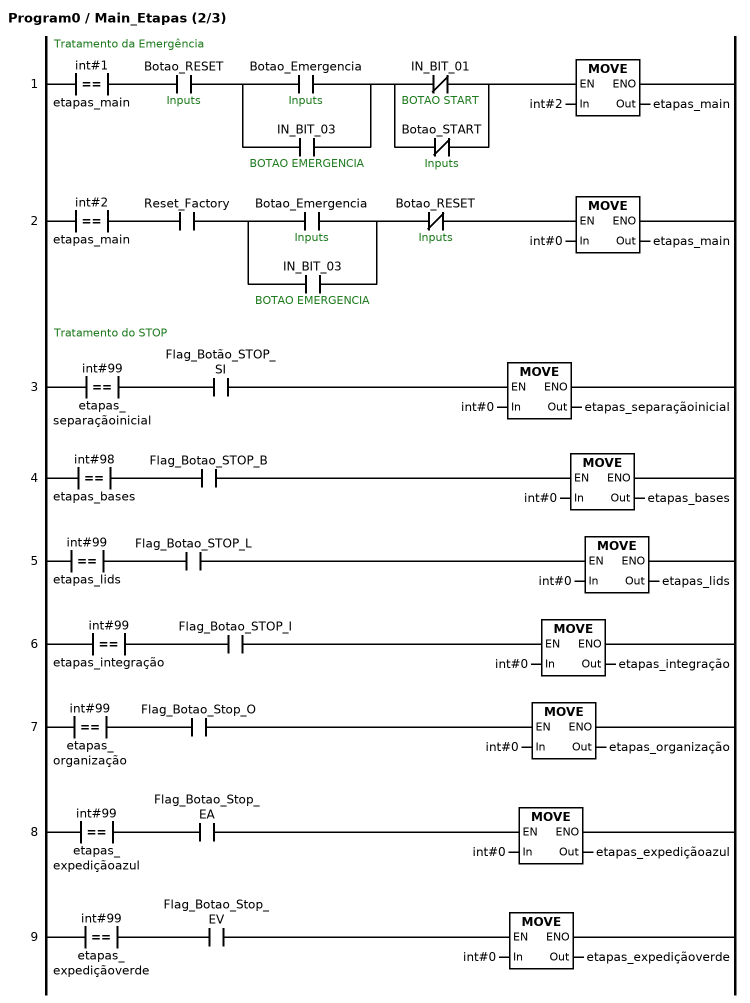
(* Rung 1: Tratamento da Emergência *)
IF (int#1 = etapas_main) AND Botao_RESET AND (Botao_Emergencia OR IN_BIT_03) AND (NOT IN_BIT_01 OR NOT Botao_START) THEN
    etapas_main := int#2;
END_IF;
(* Rung 2 *)
IF (int#2 = etapas_main) AND Reset_Factory AND (Botao_Emergencia OR IN_BIT_03) AND NOT Botao_RESET THEN
    etapas_main := int#0;
END_IF;
(* Rung 3: Tratamento do STOP *)
IF (int#99 = etapas_separaçãoinicial) AND Flag_Botão_STOP_SI THEN
    etapas_separaçãoinicial := int#0;
END_IF;
(* Rung 4 *)
IF (int#98 = etapas_bases) AND Flag_Botao_STOP_B THEN etapas_bases := int#0; END_IF;
(* Rung 5 *)
IF (int#99 = etapas_lids) AND Flag_Botao_STOP_L THEN etapas_lids := int#0; END_IF;
(* Rung 6 *)
IF (int#99 = etapas_integração) AND Flag_Botao_STOP_I THEN etapas_integração := int#0; END_IF;
(* Rung 7 *)
IF (int#99 = etapas_organização) AND Flag_Botao_Stop_O THEN etapas_organização := int#0; END_IF;
(* Rung 8 *)
IF (int#99 = etapas_expediçãoazul) AND Flag_Botao_Stop_EA THEN etapas_expediçãoazul := int#0; END_IF;
(* Rung 9 *)
IF (int#99 = etapas_expediçãoverde) AND Flag_Botao_Stop_EV THEN etapas_expediçãoverde := int#0; END_IF;

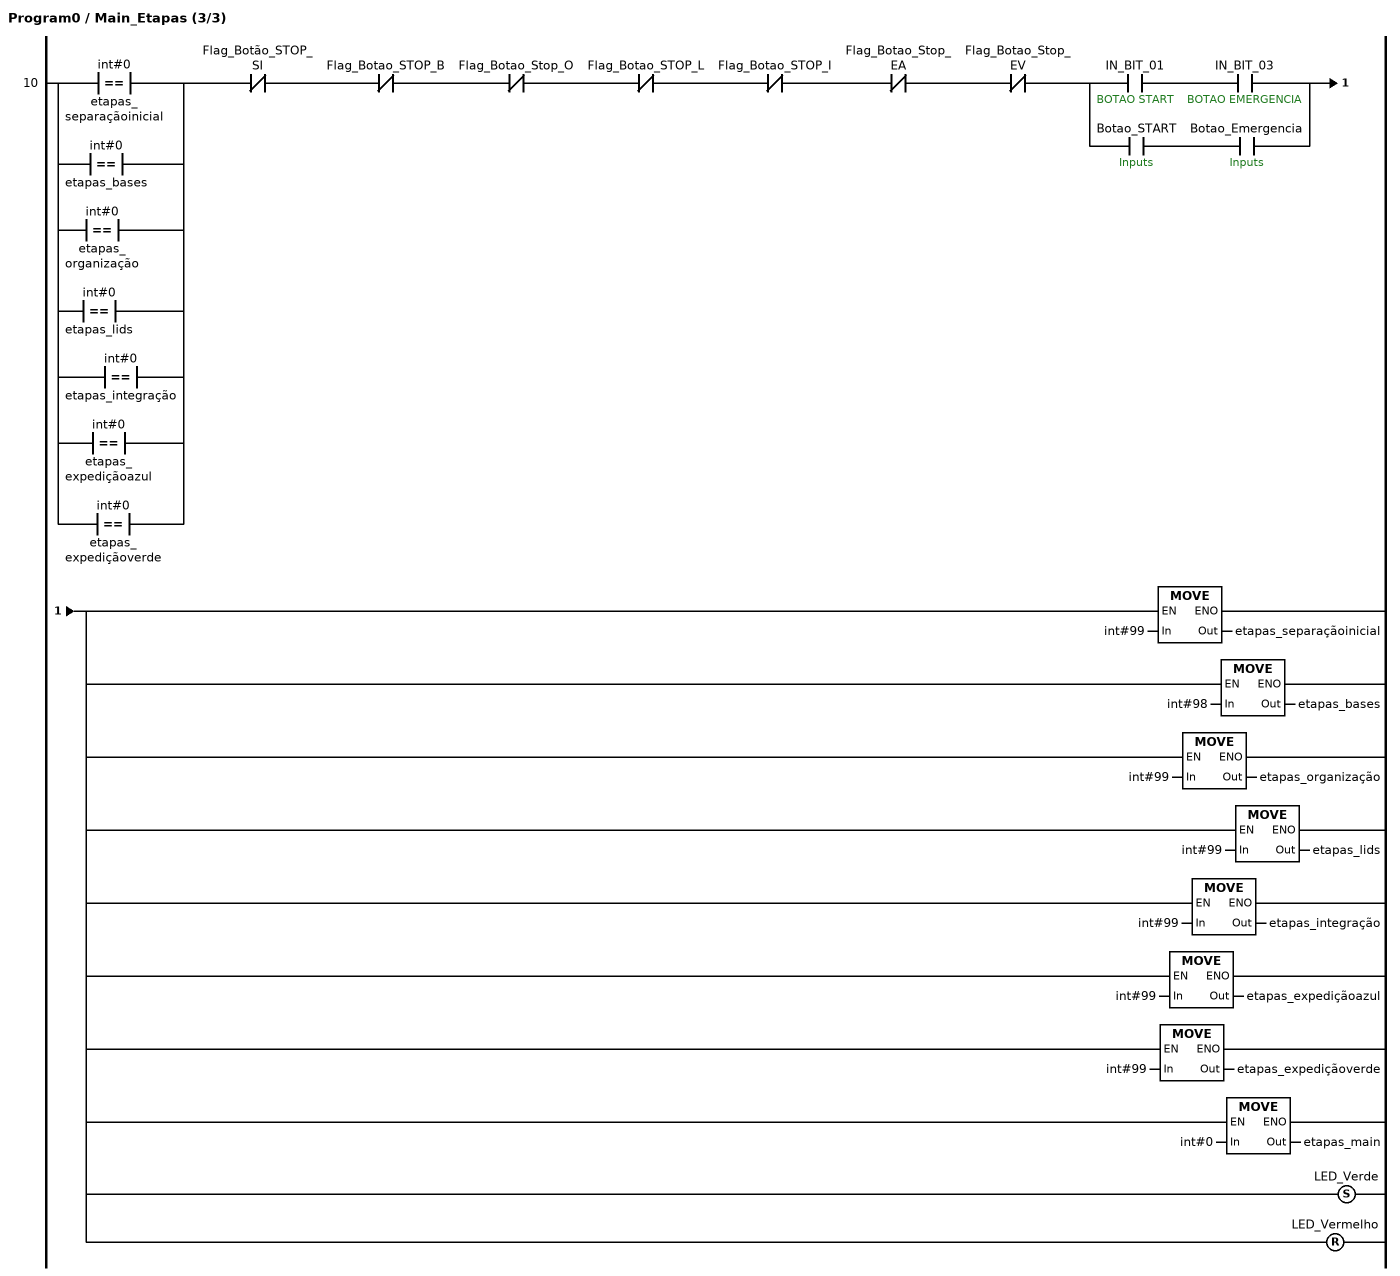
(* Rung 10 *)
_p3 := ((int#0 = etapas_separaçãoinicial) OR (int#0 = etapas_bases) OR (int#0 = etapas_organização) OR (int#0 = etapas_lids) OR (int#0 = etapas_integração) OR (int#0 = etapas_expediçãoazul) OR (int#0 = etapas_expediçãoverde)) AND NOT Flag_Botão_STOP_SI AND NOT Flag_Botao_STOP_B AND NOT Flag_Botao_Stop_O AND NOT Flag_Botao_STOP_L AND NOT Flag_Botao_STOP_I AND NOT Flag_Botao_Stop_EA AND NOT Flag_Botao_Stop_EV AND ((IN_BIT_01 AND IN_BIT_03) OR (Botao_START AND Botao_Emergencia));
IF _p3 THEN
    etapas_separaçãoinicial := int#99;
    etapas_bases := int#98;
    etapas_organização := int#99;
    etapas_lids := int#99;
    etapas_integração := int#99;
    etapas_expediçãoazul := int#99;
    etapas_expediçãoverde := int#99;
    etapas_main := int#0;
    LED_Verde := TRUE;
    LED_Vermelho := FALSE;
END_IF;

(* Section Main_Saídas: ladder, written here as Structured Text *)

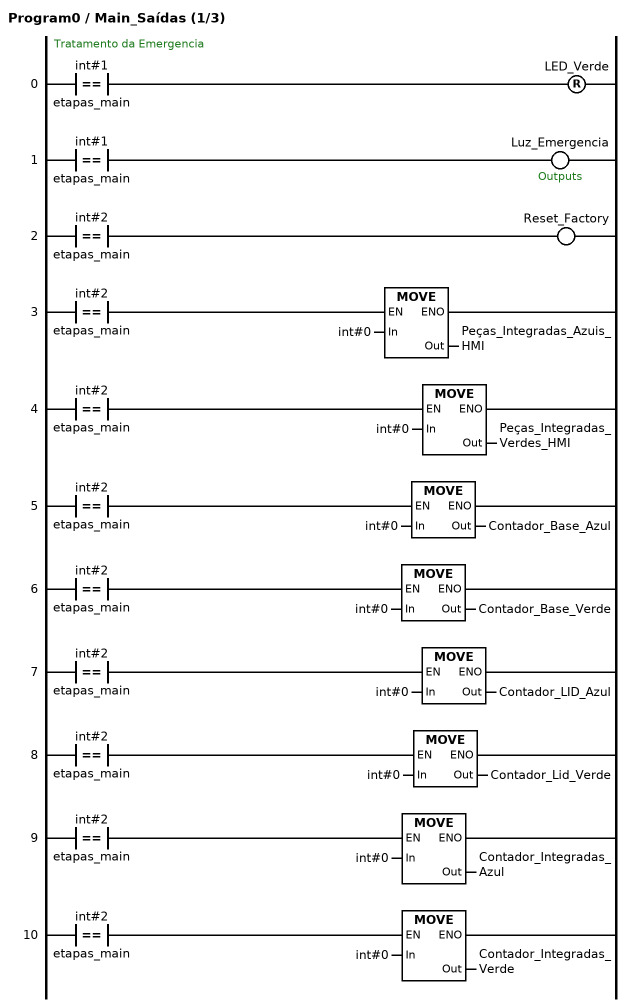
(* Rung 0: Tratamento da Emergencia *)
IF int#1 = etapas_main THEN LED_Verde := FALSE; END_IF;
(* Rung 1 *)
Luz_Emergencia := int#1 = etapas_main;
(* Rung 2 *)
Reset_Factory := int#2 = etapas_main;
(* Rung 3 *)
IF int#2 = etapas_main THEN Peças_Integradas_Azuis_HMI := int#0; END_IF;
(* Rung 4 *)
IF int#2 = etapas_main THEN Peças_Integradas_Verdes_HMI := int#0; END_IF;
(* Rung 5 *)
IF int#2 = etapas_main THEN Contador_Base_Azul := int#0; END_IF;
(* Rung 6 *)
IF int#2 = etapas_main THEN Contador_Base_Verde := int#0; END_IF;
(* Rung 7 *)
IF int#2 = etapas_main THEN Contador_LID_Azul := int#0; END_IF;
(* Rung 8 *)
IF int#2 = etapas_main THEN Contador_Lid_Verde := int#0; END_IF;
(* Rung 9 *)
IF int#2 = etapas_main THEN Contador_Integradas_Azul := int#0; END_IF;
(* Rung 10 *)
IF int#2 = etapas_main THEN Contador_Integradas_Verde := int#0; END_IF;

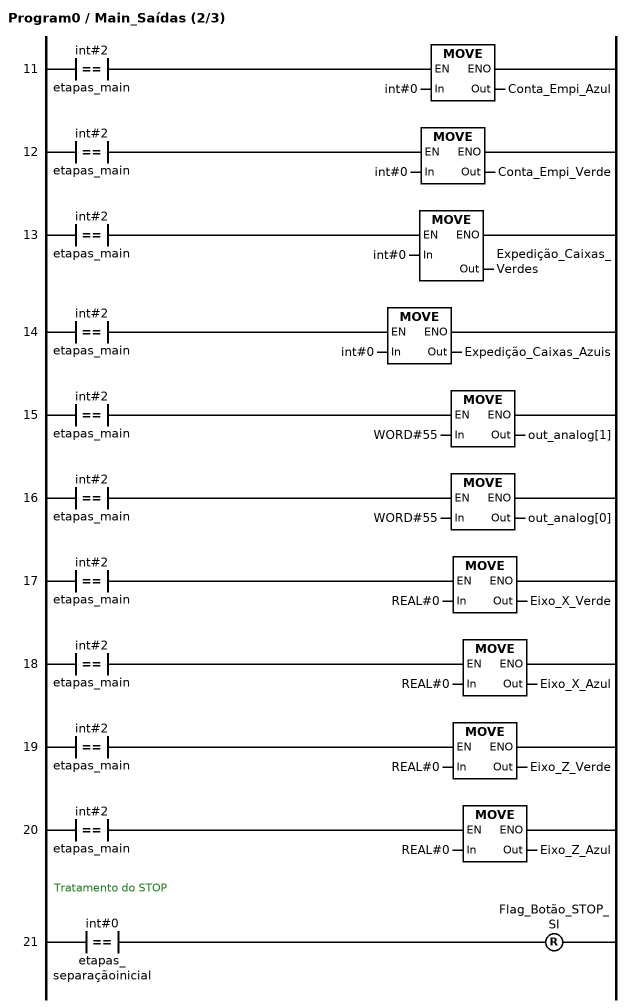
(* Rung 11 *)
IF int#2 = etapas_main THEN Conta_Empi_Azul := int#0; END_IF;
(* Rung 12 *)
IF int#2 = etapas_main THEN Conta_Empi_Verde := int#0; END_IF;
(* Rung 13 *)
IF int#2 = etapas_main THEN Expedição_Caixas_Verdes := int#0; END_IF;
(* Rung 14 *)
IF int#2 = etapas_main THEN Expedição_Caixas_Azuis := int#0; END_IF;
(* Rung 15 *)
IF int#2 = etapas_main THEN out_analog[1] := WORD#55; END_IF;
(* Rung 16 *)
IF int#2 = etapas_main THEN out_analog[0] := WORD#55; END_IF;
(* Rung 17 *)
IF int#2 = etapas_main THEN Eixo_X_Verde := REAL#0; END_IF;
(* Rung 18 *)
IF int#2 = etapas_main THEN Eixo_X_Azul := REAL#0; END_IF;
(* Rung 19 *)
IF int#2 = etapas_main THEN Eixo_Z_Verde := REAL#0; END_IF;
(* Rung 20 *)
IF int#2 = etapas_main THEN Eixo_Z_Azul := REAL#0; END_IF;
(* Rung 21: Tratamento do STOP *)
IF int#0 = etapas_separaçãoinicial THEN Flag_Botão_STOP_SI := FALSE; END_IF;

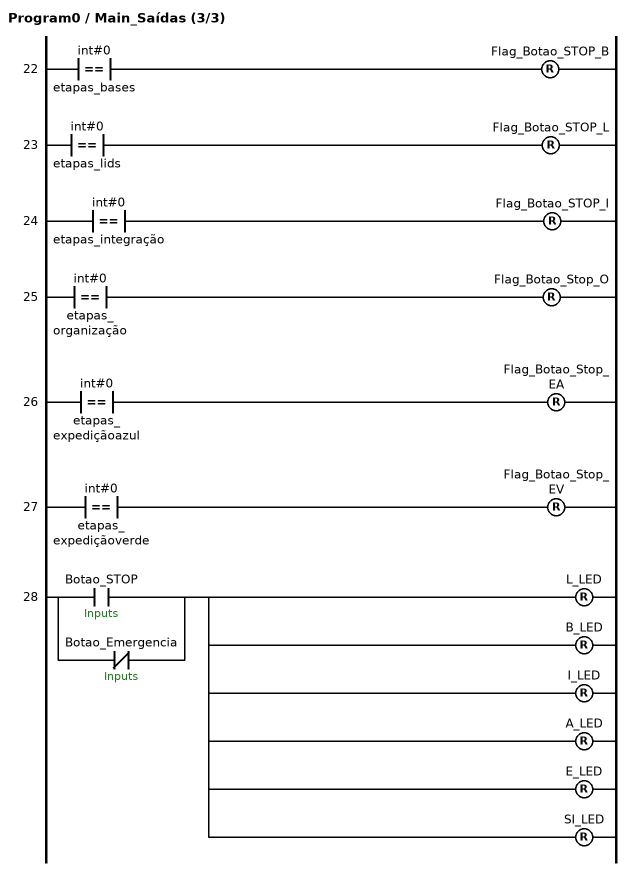
(* Rung 22 *)
IF int#0 = etapas_bases THEN Flag_Botao_STOP_B := FALSE; END_IF;
(* Rung 23 *)
IF int#0 = etapas_lids THEN Flag_Botao_STOP_L := FALSE; END_IF;
(* Rung 24 *)
IF int#0 = etapas_integração THEN Flag_Botao_STOP_I := FALSE; END_IF;
(* Rung 25 *)
IF int#0 = etapas_organização THEN Flag_Botao_Stop_O := FALSE; END_IF;
(* Rung 26 *)
IF int#0 = etapas_expediçãoazul THEN Flag_Botao_Stop_EA := FALSE; END_IF;
(* Rung 27 *)
IF int#0 = etapas_expediçãoverde THEN Flag_Botao_Stop_EV := FALSE; END_IF;
(* Rung 28 *)
IF Botao_STOP OR NOT Botao_Emergencia THEN
    L_LED := FALSE;
    B_LED := FALSE;
    I_LED := FALSE;
    A_LED := FALSE;
    E_LED := FALSE;
    SI_LED := FALSE;
END_IF;

(* Section Input_Fisico: ladder, written here as Structured Text *)

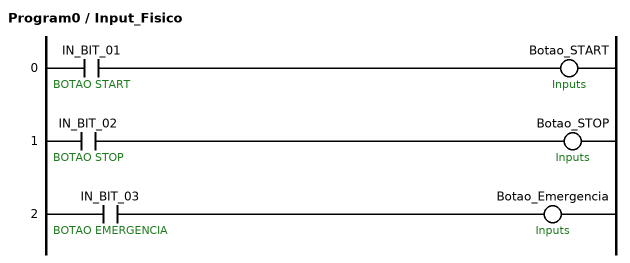
(* Rung 0 *)
Botao_START := IN_BIT_01;
(* Rung 1 *)
Botao_STOP := IN_BIT_02;
(* Rung 2 *)
Botao_Emergencia := IN_BIT_03;

(* Section Output_Fisico: ladder, written here as Structured Text *)

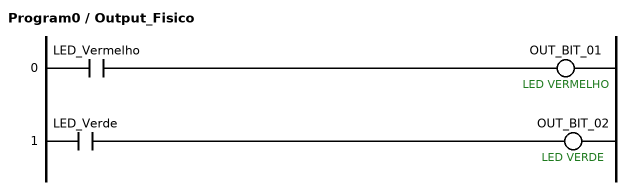
(* Rung 0 *)
OUT_BIT_01 := LED_Vermelho;
(* Rung 1 *)
OUT_BIT_02 := LED_Verde;

(* Section Input_Dig: ladder, written here as Structured Text *)

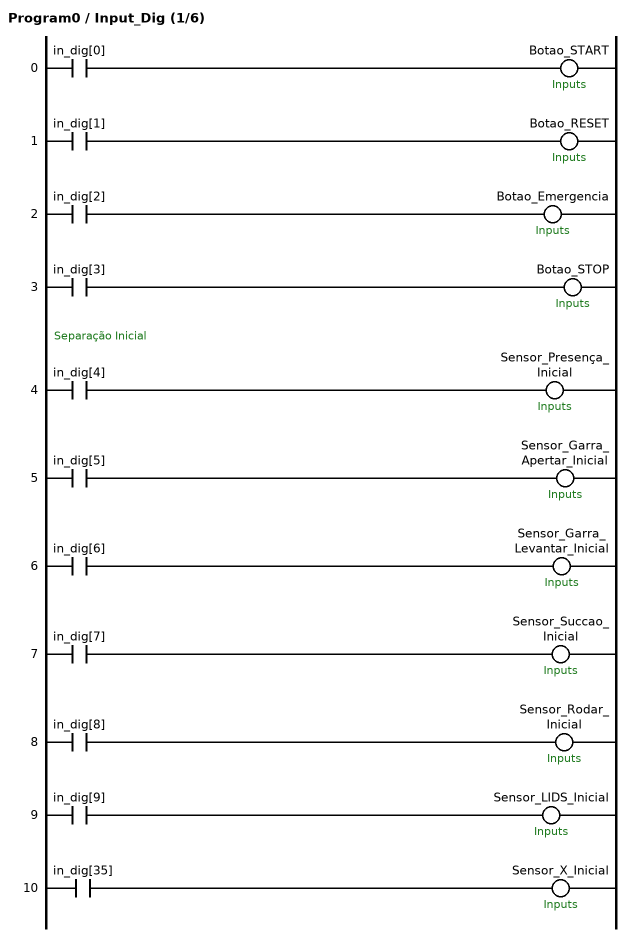
(* Rung 0 *)
Botao_START := in_dig[0];
(* Rung 1 *)
Botao_RESET := in_dig[1];
(* Rung 2 *)
Botao_Emergencia := in_dig[2];
(* Rung 3 *)
Botao_STOP := in_dig[3];
(* Rung 4: Separação Inicial *)
Sensor_Presença_Inicial := in_dig[4];
(* Rung 5 *)
Sensor_Garra_Apertar_Inicial := in_dig[5];
(* Rung 6 *)
Sensor_Garra_Levantar_Inicial := in_dig[6];
(* Rung 7 *)
Sensor_Succao_Inicial := in_dig[7];
(* Rung 8 *)
Sensor_Rodar_Inicial := in_dig[8];
(* Rung 9 *)
Sensor_LIDS_Inicial := in_dig[9];
(* Rung 10 *)
Sensor_X_Inicial := in_dig[35];

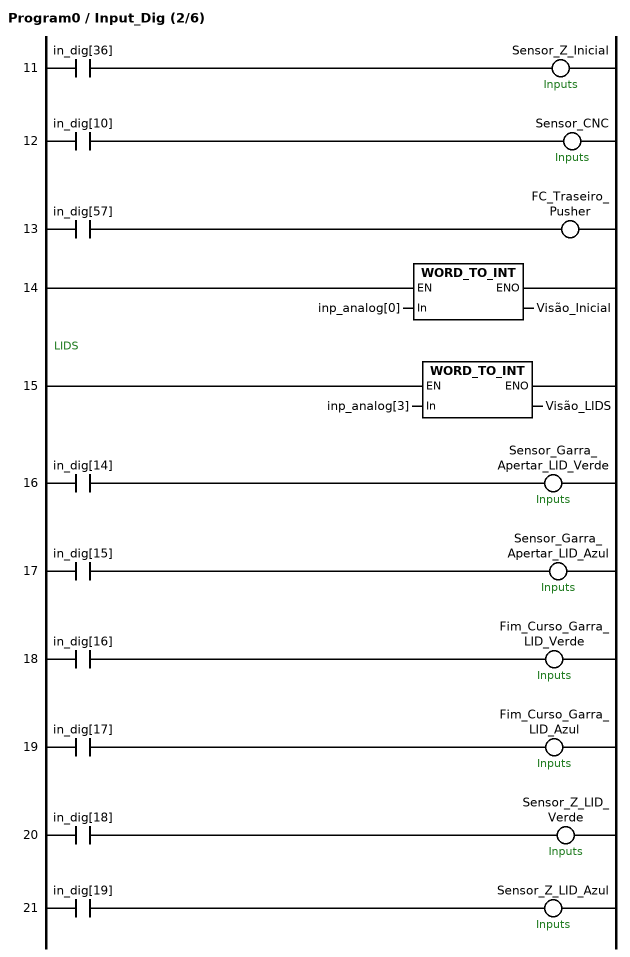
(* Rung 11 *)
Sensor_Z_Inicial := in_dig[36];
(* Rung 12 *)
Sensor_CNC := in_dig[10];
(* Rung 13 *)
FC_Traseiro_Pusher := in_dig[57];
(* Rung 14 *)
Visão_Inicial := WORD_TO_INT(In := inp_analog[0]);
(* Rung 15: LIDS *)
Visão_LIDS := WORD_TO_INT(In := inp_analog[3]);
(* Rung 16 *)
Sensor_Garra_Apertar_LID_Verde := in_dig[14];
(* Rung 17 *)
Sensor_Garra_Apertar_LID_Azul := in_dig[15];
(* Rung 18 *)
Fim_Curso_Garra_LID_Verde := in_dig[16];
(* Rung 19 *)
Fim_Curso_Garra_LID_Azul := in_dig[17];
(* Rung 20 *)
Sensor_Z_LID_Verde := in_dig[18];
(* Rung 21 *)
Sensor_Z_LID_Azul := in_dig[19];

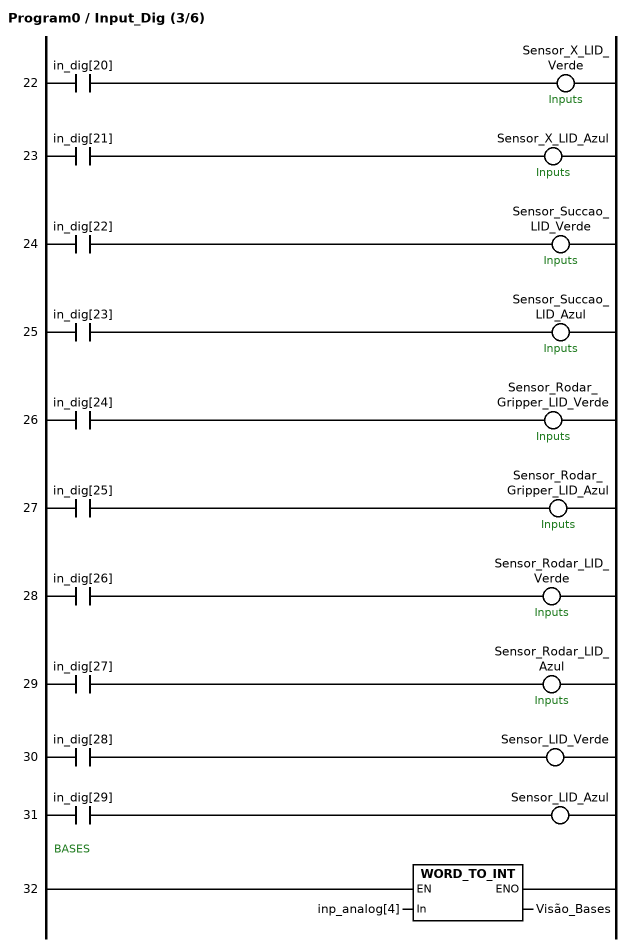
(* Rung 22 *)
Sensor_X_LID_Verde := in_dig[20];
(* Rung 23 *)
Sensor_X_LID_Azul := in_dig[21];
(* Rung 24 *)
Sensor_Succao_LID_Verde := in_dig[22];
(* Rung 25 *)
Sensor_Succao_LID_Azul := in_dig[23];
(* Rung 26 *)
Sensor_Rodar_Gripper_LID_Verde := in_dig[24];
(* Rung 27 *)
Sensor_Rodar_Gripper_LID_Azul := in_dig[25];
(* Rung 28 *)
Sensor_Rodar_LID_Verde := in_dig[26];
(* Rung 29 *)
Sensor_Rodar_LID_Azul := in_dig[27];
(* Rung 30 *)
Sensor_LID_Verde := in_dig[28];
(* Rung 31 *)
Sensor_LID_Azul := in_dig[29];
(* Rung 32: BASES *)
Visão_Bases := WORD_TO_INT(In := inp_analog[4]);

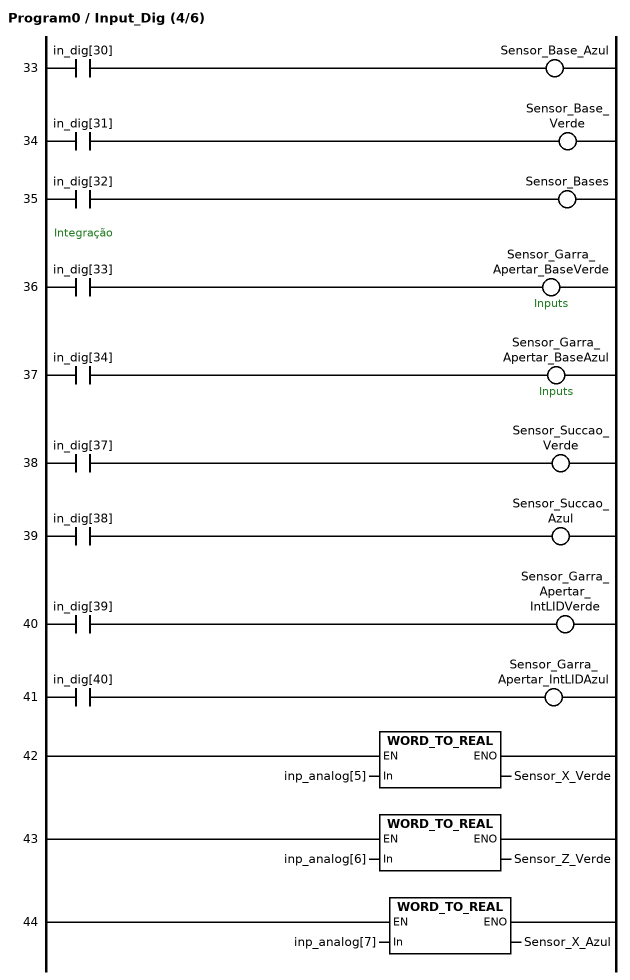
(* Rung 33 *)
Sensor_Base_Azul := in_dig[30];
(* Rung 34 *)
Sensor_Base_Verde := in_dig[31];
(* Rung 35 *)
Sensor_Bases := in_dig[32];
(* Rung 36: Integração *)
Sensor_Garra_Apertar_BaseVerde := in_dig[33];
(* Rung 37 *)
Sensor_Garra_Apertar_BaseAzul := in_dig[34];
(* Rung 38 *)
Sensor_Succao_Verde := in_dig[37];
(* Rung 39 *)
Sensor_Succao_Azul := in_dig[38];
(* Rung 40 *)
Sensor_Garra_Apertar_IntLIDVerde := in_dig[39];
(* Rung 41 *)
Sensor_Garra_Apertar_IntLIDAzul := in_dig[40];
(* Rung 42 *)
Sensor_X_Verde := WORD_TO_REAL(In := inp_analog[5]);
(* Rung 43 *)
Sensor_Z_Verde := WORD_TO_REAL(In := inp_analog[6]);
(* Rung 44 *)
Sensor_X_Azul := WORD_TO_REAL(In := inp_analog[7]);

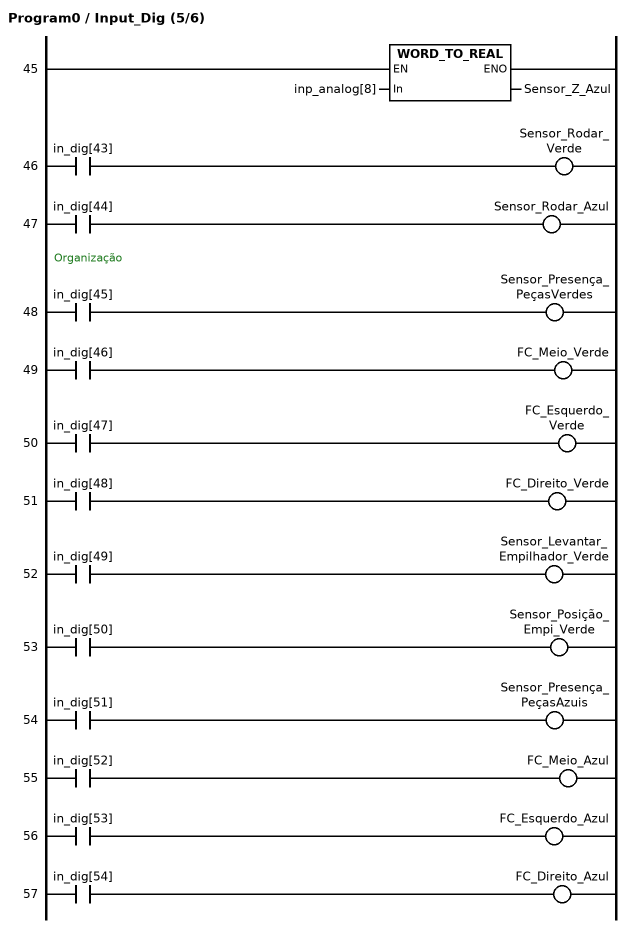
(* Rung 45 *)
Sensor_Z_Azul := WORD_TO_REAL(In := inp_analog[8]);
(* Rung 46 *)
Sensor_Rodar_Verde := in_dig[43];
(* Rung 47 *)
Sensor_Rodar_Azul := in_dig[44];
(* Rung 48: Organização *)
Sensor_Presença_PeçasVerdes := in_dig[45];
(* Rung 49 *)
FC_Meio_Verde := in_dig[46];
(* Rung 50 *)
FC_Esquerdo_Verde := in_dig[47];
(* Rung 51 *)
FC_Direito_Verde := in_dig[48];
(* Rung 52 *)
Sensor_Levantar_Empilhador_Verde := in_dig[49];
(* Rung 53 *)
Sensor_Posição_Empi_Verde := in_dig[50];
(* Rung 54 *)
Sensor_Presença_PeçasAzuis := in_dig[51];
(* Rung 55 *)
FC_Meio_Azul := in_dig[52];
(* Rung 56 *)
FC_Esquerdo_Azul := in_dig[53];
(* Rung 57 *)
FC_Direito_Azul := in_dig[54];

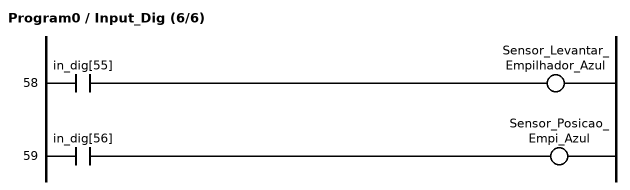
(* Rung 58 *)
Sensor_Levantar_Empilhador_Azul := in_dig[55];
(* Rung 59 *)
Sensor_Posicao_Empi_Azul := in_dig[56];

(* Section Output_Dig: ladder, written here as Structured Text *)

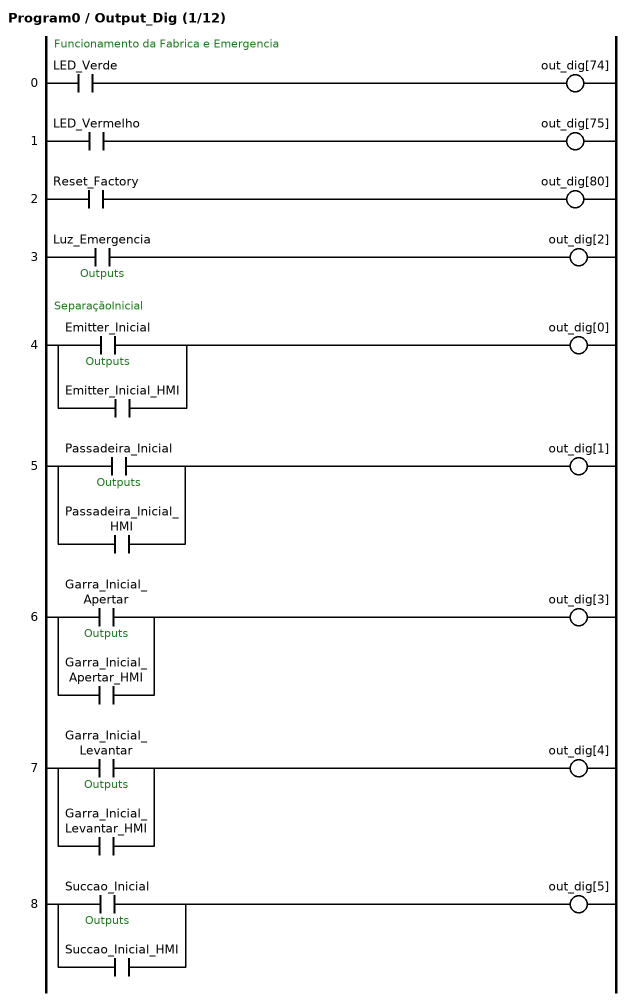
(* Rung 0: Funcionamento da Fabrica e Emergencia *)
out_dig[74] := LED_Verde;
(* Rung 1 *)
out_dig[75] := LED_Vermelho;
(* Rung 2 *)
out_dig[80] := Reset_Factory;
(* Rung 3 *)
out_dig[2] := Luz_Emergencia;
(* Rung 4: SeparaçãoInicial *)
out_dig[0] := Emitter_Inicial OR Emitter_Inicial_HMI;
(* Rung 5 *)
out_dig[1] := Passadeira_Inicial OR Passadeira_Inicial_HMI;
(* Rung 6 *)
out_dig[3] := Garra_Inicial_Apertar OR Garra_Inicial_Apertar_HMI;
(* Rung 7 *)
out_dig[4] := Garra_Inicial_Levantar OR Garra_Inicial_Levantar_HMI;
(* Rung 8 *)
out_dig[5] := Succao_Inicial OR Succao_Inicial_HMI;

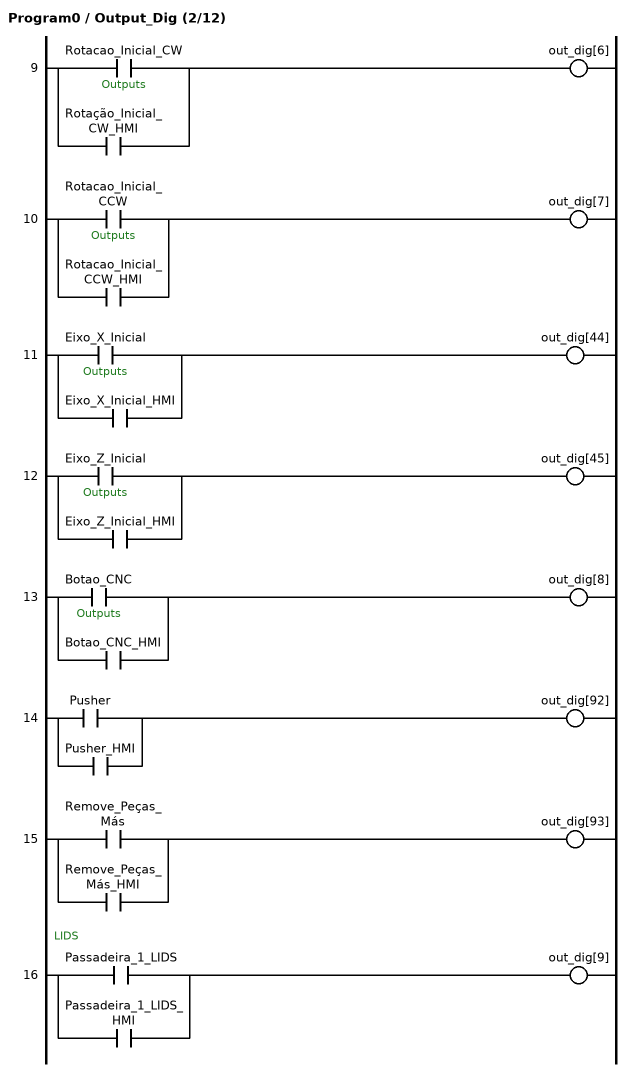
(* Rung 9 *)
out_dig[6] := Rotacao_Inicial_CW OR Rotação_Inicial_CW_HMI;
(* Rung 10 *)
out_dig[7] := Rotacao_Inicial_CCW OR Rotacao_Inicial_CCW_HMI;
(* Rung 11 *)
out_dig[44] := Eixo_X_Inicial OR Eixo_X_Inicial_HMI;
(* Rung 12 *)
out_dig[45] := Eixo_Z_Inicial OR Eixo_Z_Inicial_HMI;
(* Rung 13 *)
out_dig[8] := Botao_CNC OR Botao_CNC_HMI;
(* Rung 14 *)
out_dig[92] := Pusher OR Pusher_HMI;
(* Rung 15 *)
out_dig[93] := Remove_Peças_Más OR Remove_Peças_Más_HMI;
(* Rung 16: LIDS *)
out_dig[9] := Passadeira_1_LIDS OR Passadeira_1_LIDS_HMI;

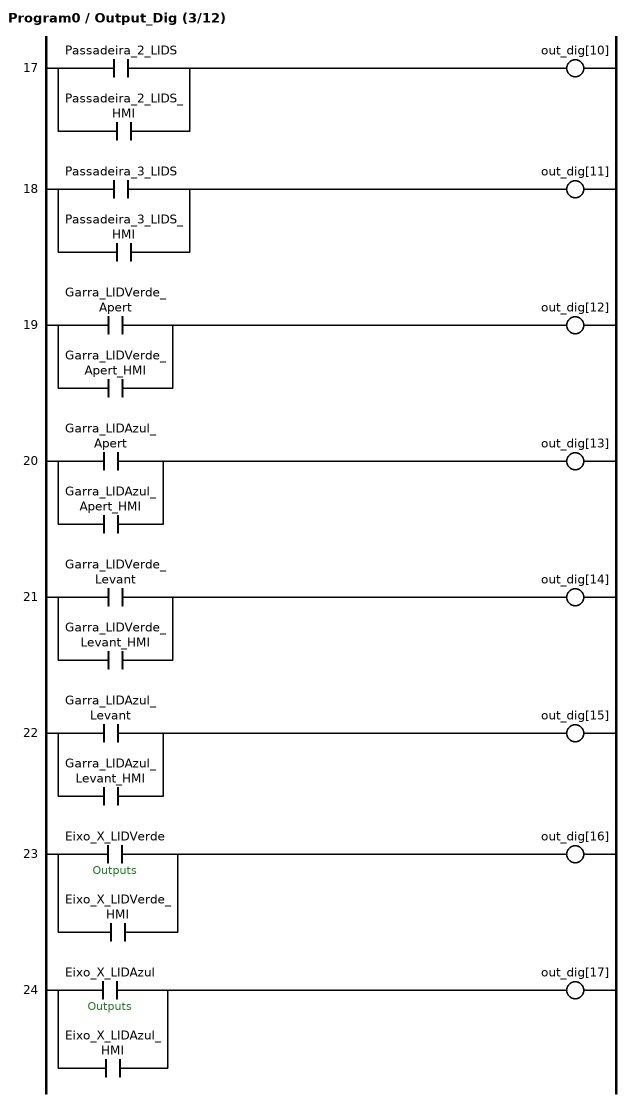
(* Rung 17 *)
out_dig[10] := Passadeira_2_LIDS OR Passadeira_2_LIDS_HMI;
(* Rung 18 *)
out_dig[11] := Passadeira_3_LIDS OR Passadeira_3_LIDS_HMI;
(* Rung 19 *)
out_dig[12] := Garra_LIDVerde_Apert OR Garra_LIDVerde_Apert_HMI;
(* Rung 20 *)
out_dig[13] := Garra_LIDAzul_Apert OR Garra_LIDAzul_Apert_HMI;
(* Rung 21 *)
out_dig[14] := Garra_LIDVerde_Levant OR Garra_LIDVerde_Levant_HMI;
(* Rung 22 *)
out_dig[15] := Garra_LIDAzul_Levant OR Garra_LIDAzul_Levant_HMI;
(* Rung 23 *)
out_dig[16] := Eixo_X_LIDVerde OR Eixo_X_LIDVerde_HMI;
(* Rung 24 *)
out_dig[17] := Eixo_X_LIDAzul OR Eixo_X_LIDAzul_HMI;

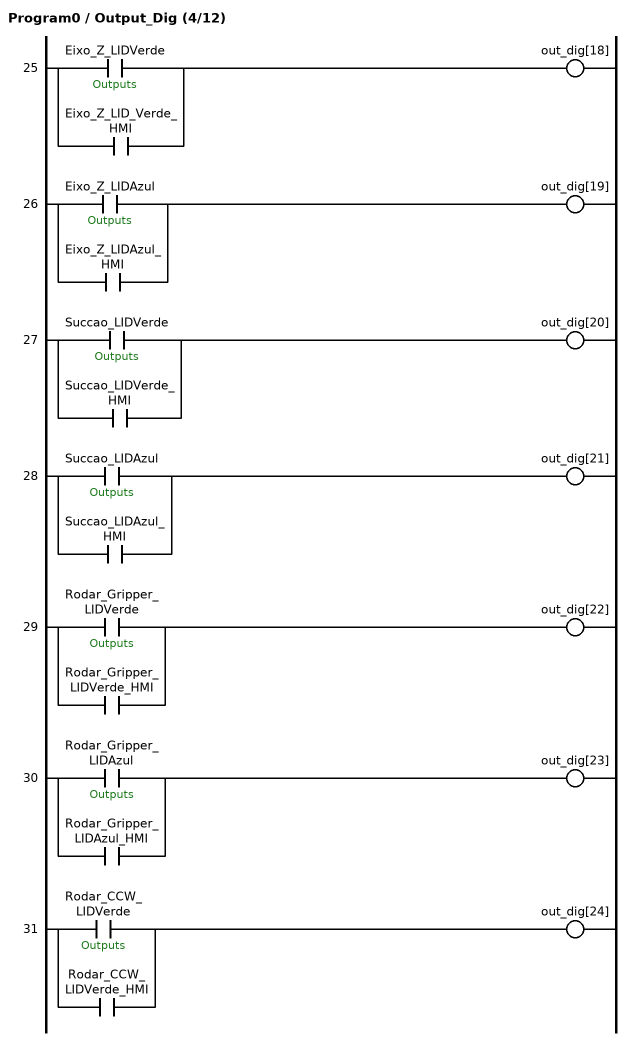
(* Rung 25 *)
out_dig[18] := Eixo_Z_LIDVerde OR Eixo_Z_LID_Verde_HMI;
(* Rung 26 *)
out_dig[19] := Eixo_Z_LIDAzul OR Eixo_Z_LIDAzul_HMI;
(* Rung 27 *)
out_dig[20] := Succao_LIDVerde OR Succao_LIDVerde_HMI;
(* Rung 28 *)
out_dig[21] := Succao_LIDAzul OR Succao_LIDAzul_HMI;
(* Rung 29 *)
out_dig[22] := Rodar_Gripper_LIDVerde OR Rodar_Gripper_LIDVerde_HMI;
(* Rung 30 *)
out_dig[23] := Rodar_Gripper_LIDAzul OR Rodar_Gripper_LIDAzul_HMI;
(* Rung 31 *)
out_dig[24] := Rodar_CCW_LIDVerde OR Rodar_CCW_LIDVerde_HMI;

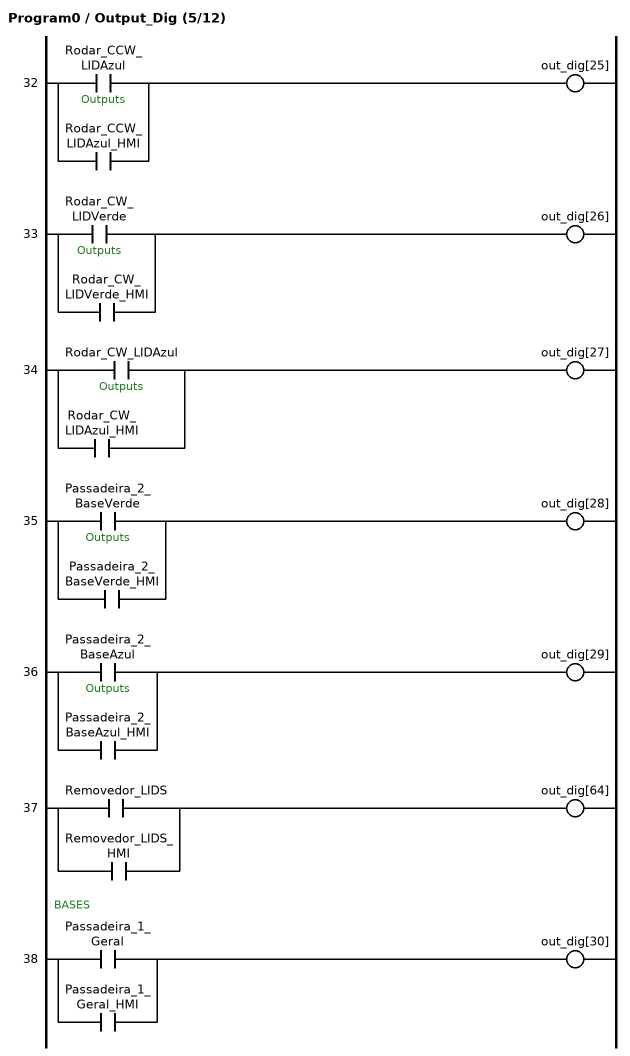
(* Rung 32 *)
out_dig[25] := Rodar_CCW_LIDAzul OR Rodar_CCW_LIDAzul_HMI;
(* Rung 33 *)
out_dig[26] := Rodar_CW_LIDVerde OR Rodar_CW_LIDVerde_HMI;
(* Rung 34 *)
out_dig[27] := Rodar_CW_LIDAzul OR Rodar_CW_LIDAzul_HMI;
(* Rung 35 *)
out_dig[28] := Passadeira_2_BaseVerde OR Passadeira_2_BaseVerde_HMI;
(* Rung 36 *)
out_dig[29] := Passadeira_2_BaseAzul OR Passadeira_2_BaseAzul_HMI;
(* Rung 37 *)
out_dig[64] := Removedor_LIDS OR Removedor_LIDS_HMI;
(* Rung 38: BASES *)
out_dig[30] := Passadeira_1_Geral OR Passadeira_1_Geral_HMI;

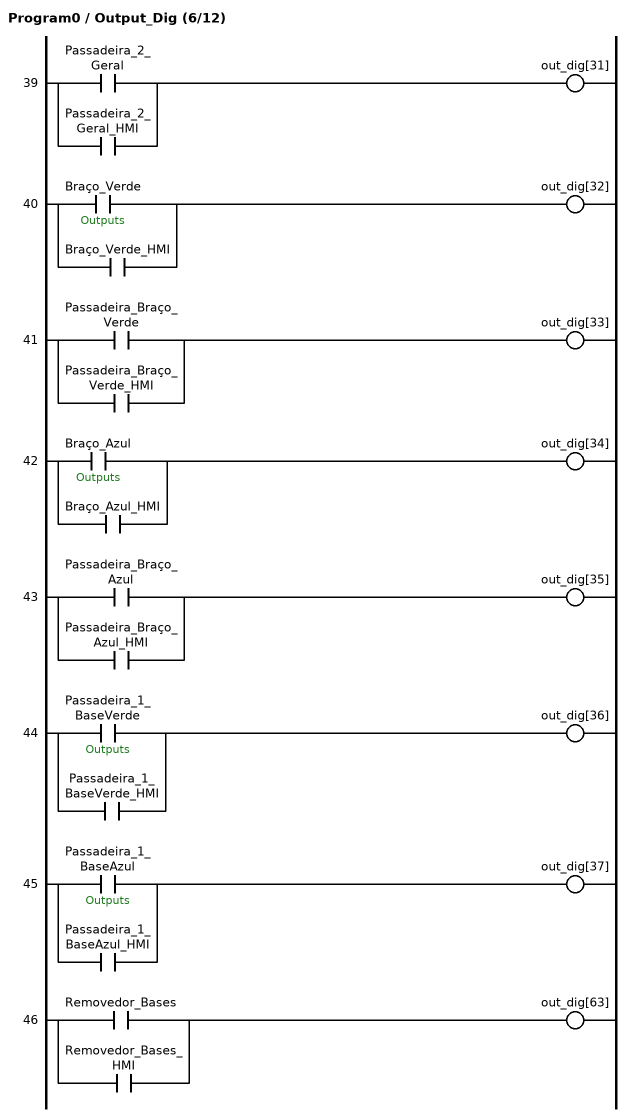
(* Rung 39 *)
out_dig[31] := Passadeira_2_Geral OR Passadeira_2_Geral_HMI;
(* Rung 40 *)
out_dig[32] := Braço_Verde OR Braço_Verde_HMI;
(* Rung 41 *)
out_dig[33] := Passadeira_Braço_Verde OR Passadeira_Braço_Verde_HMI;
(* Rung 42 *)
out_dig[34] := Braço_Azul OR Braço_Azul_HMI;
(* Rung 43 *)
out_dig[35] := Passadeira_Braço_Azul OR Passadeira_Braço_Azul_HMI;
(* Rung 44 *)
out_dig[36] := Passadeira_1_BaseVerde OR Passadeira_1_BaseVerde_HMI;
(* Rung 45 *)
out_dig[37] := Passadeira_1_BaseAzul OR Passadeira_1_BaseAzul_HMI;
(* Rung 46 *)
out_dig[63] := Removedor_Bases OR Removedor_Bases_HMI;

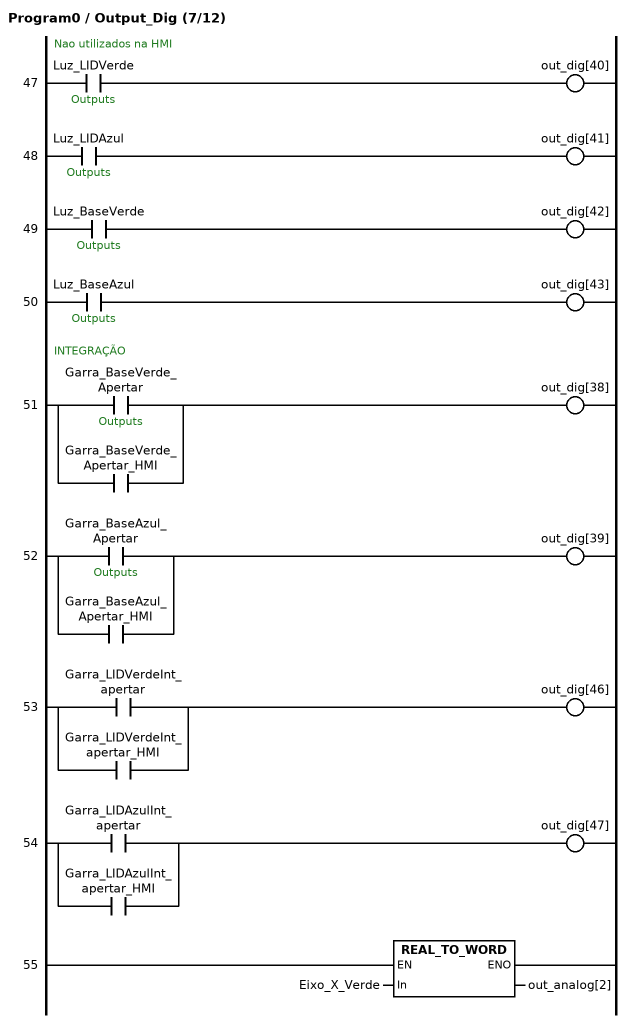
(* Rung 47: Nao utilizados na HMI *)
out_dig[40] := Luz_LIDVerde;
(* Rung 48 *)
out_dig[41] := Luz_LIDAzul;
(* Rung 49 *)
out_dig[42] := Luz_BaseVerde;
(* Rung 50 *)
out_dig[43] := Luz_BaseAzul;
(* Rung 51: INTEGRAÇÃO *)
out_dig[38] := Garra_BaseVerde_Apertar OR Garra_BaseVerde_Apertar_HMI;
(* Rung 52 *)
out_dig[39] := Garra_BaseAzul_Apertar OR Garra_BaseAzul_Apertar_HMI;
(* Rung 53 *)
out_dig[46] := Garra_LIDVerdeInt_apertar OR Garra_LIDVerdeInt_apertar_HMI;
(* Rung 54 *)
out_dig[47] := Garra_LIDAzulInt_apertar OR Garra_LIDAzulInt_apertar_HMI;
(* Rung 55 *)
out_analog[2] := REAL_TO_WORD(In := Eixo_X_Verde);

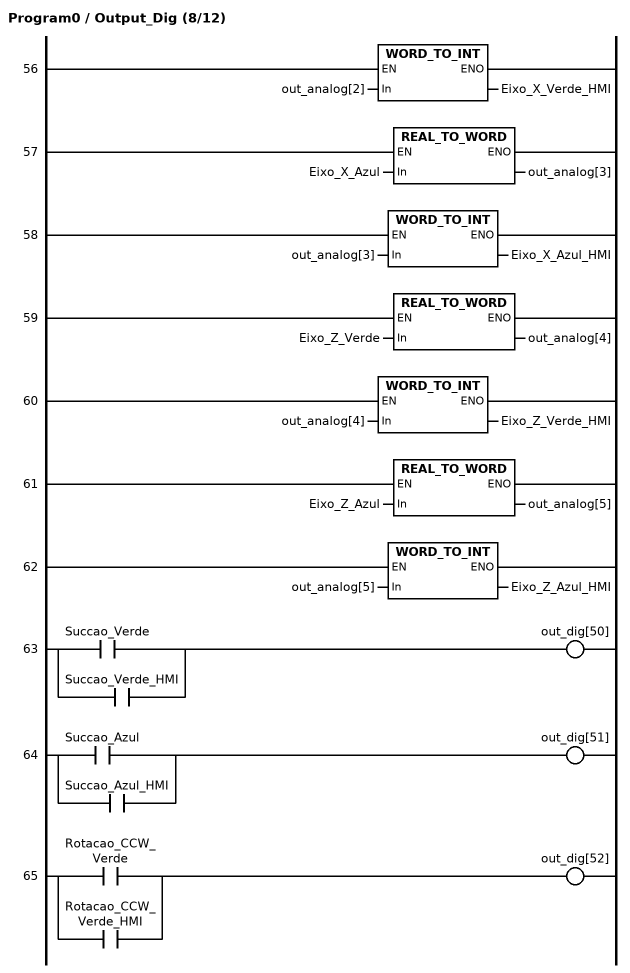
(* Rung 56 *)
Eixo_X_Verde_HMI := WORD_TO_INT(In := out_analog[2]);
(* Rung 57 *)
out_analog[3] := REAL_TO_WORD(In := Eixo_X_Azul);
(* Rung 58 *)
Eixo_X_Azul_HMI := WORD_TO_INT(In := out_analog[3]);
(* Rung 59 *)
out_analog[4] := REAL_TO_WORD(In := Eixo_Z_Verde);
(* Rung 60 *)
Eixo_Z_Verde_HMI := WORD_TO_INT(In := out_analog[4]);
(* Rung 61 *)
out_analog[5] := REAL_TO_WORD(In := Eixo_Z_Azul);
(* Rung 62 *)
Eixo_Z_Azul_HMI := WORD_TO_INT(In := out_analog[5]);
(* Rung 63 *)
out_dig[50] := Succao_Verde OR Succao_Verde_HMI;
(* Rung 64 *)
out_dig[51] := Succao_Azul OR Succao_Azul_HMI;
(* Rung 65 *)
out_dig[52] := Rotacao_CCW_Verde OR Rotacao_CCW_Verde_HMI;

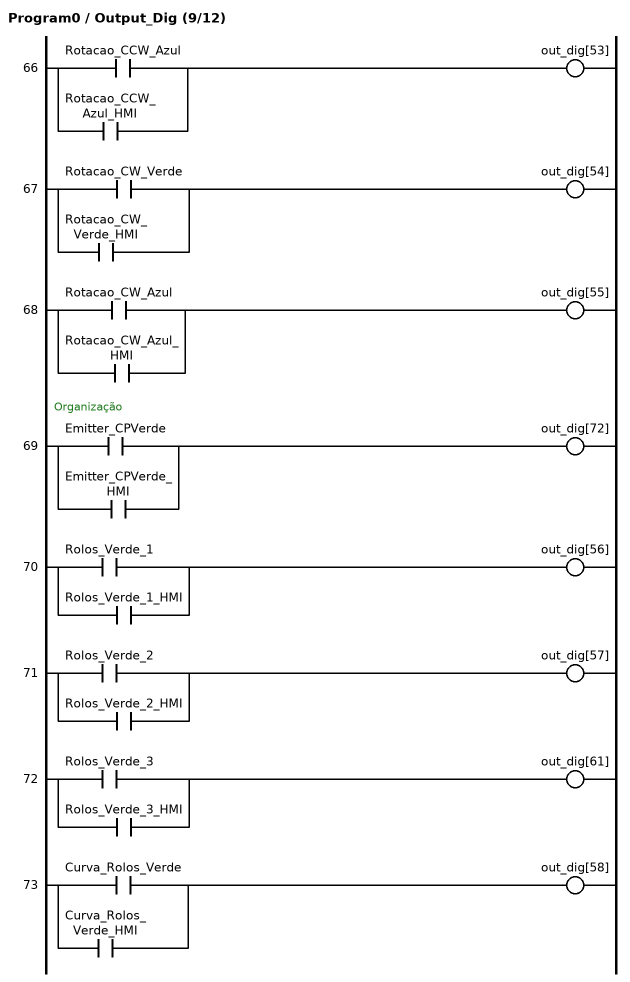
(* Rung 66 *)
out_dig[53] := Rotacao_CCW_Azul OR Rotacao_CCW_Azul_HMI;
(* Rung 67 *)
out_dig[54] := Rotacao_CW_Verde OR Rotacao_CW_Verde_HMI;
(* Rung 68 *)
out_dig[55] := Rotacao_CW_Azul OR Rotacao_CW_Azul_HMI;
(* Rung 69: Organização *)
out_dig[72] := Emitter_CPVerde OR Emitter_CPVerde_HMI;
(* Rung 70 *)
out_dig[56] := Rolos_Verde_1 OR Rolos_Verde_1_HMI;
(* Rung 71 *)
out_dig[57] := Rolos_Verde_2 OR Rolos_Verde_2_HMI;
(* Rung 72 *)
out_dig[61] := Rolos_Verde_3 OR Rolos_Verde_3_HMI;
(* Rung 73 *)
out_dig[58] := Curva_Rolos_Verde OR Curva_Rolos_Verde_HMI;

